LIN {X 0,Y 403.759,Z 485.319,A -85,B 0,C 180,E1 -11073.792,E2 -11073.792} C_VEL
LIN {X 0,Y 400.892,Z 485.679,A -85,B 0,C 180,E1 -11075.141,E2 -11075.141} C_VEL
LIN {X 0,Y 398.47,Z 485.978,A -85,B 0,C 180,E1 -11076.231,E2 -11076.231} C_VEL
LIN {X 0,Y 397.442,Z 486.102,A -85,B 0,C 180,E1 -11077.075,E2 -11077.075} C_VEL
LIN {X 0,Y 397.364,Z 486.11,A -85,B 0,C 180,E1 -11077.36,E2 -11077.36} C_VEL
LIN {X 0,Y 397.201,Z 486.134,A -85,B 0,C 180,E1 -11081.223,E2 -11081.223} C_VEL
LIN {X 0,Y 397.178,Z 486.132,A -85,B 0,C 180,E1 -11084.343,E2 -11084.343} C_VEL
LIN {X 0,Y 397.176,Z 486.138,A -85,B 0,C 180,E1 -11087.507,E2 -11087.507} C_VEL
LIN {X 0,Y 397.11,Z 486.141,A -85,B 0,C 180,E1 -11090.73,E2 -11090.73} C_VEL
LIN {X 0,Y 397.134,Z 486.138,A -85,B 0,C 180,E1 -11094.018,E2 -11094.018} C_VEL
LIN {X 0,Y 397.196,Z 486.137,A -85,B 0,C 180,E1 -11097.39,E2 -11097.39} C_VEL
LIN {X 0,Y 397.08,Z 486.146,A -85,B 0,C 180,E1 -11100.882,E2 -11100.882} C_VEL
LIN {X 0,Y 397.127,Z 486.138,A -85,B 0,C 180,E1 -11104.493,E2 -11104.493} C_VEL
LIN {X 0,Y 397.105,Z 486.141,A -85,B 0,C 180,E1 -11108.275,E2 -11108.275} C_VEL
LIN {X 0,Y 397.092,Z 486.145,A -85,B 0,C 180,E1 -11110.909,E2 -11110.909} C_VEL
LIN {X 0,Y 397.105,Z 486.144,A -85,B 0,C 180,E1 -11113.648,E2 -11113.648} C_VEL
LIN {X 0,Y 397.103,Z 486.141,A -85,B 0,C 180,E1 -11116.521,E2 -11116.521} C_VEL
LIN {X 0,Y 397.115,Z 486.14,A -85,B 0,C 180,E1 -11120.423,E2 -11120.423} C_VEL
LIN {X 0,Y 397.11,Z 486.14,A -85,B 0,C 180,E1 -11124.266,E2 -11124.266} C_VEL
LIN {X 0,Y 397.116,Z 486.141,A -85,B 0,C 180,E1 -11126.727,E2 -11126.727} C_VEL
LIN {X 0,Y 397.188,Z 486.311,A -85,B 0,C 180,E1 -11130.065,E2 -11130.065} C_VEL
LIN {X 0,Y 400.62,Z 501.643,A -85,B 0,C 180,E1 -11132.863,E2 -11132.863} C_VEL
LIN {X 0,Y 401.755,Z 508.389,A -85,B 0,C 180,E1 -11134.066,E2 -11134.066} C_VEL
LIN {X 0,Y 400.796,Z 526.433,A -85,B 0,C 180,E1 -11137.036,E2 -11137.036} C_VEL
LIN {X 0,Y 399.909,Z 544.238,A -85,B 0,C 180,E1 -11139.959,E2 -11139.959} C_VEL
LIN {X 0,Y 399.783,Z 547.353,A -85,B 0,C 180,E1 -11140.471,E2 -11140.471} C_VEL
LIN {X 0,Y 402.807,Z 568.009,A -85,B 0,C 180,E1 -11141.071,E2 -11141.071} C_VEL
LIN {X 0,Y 401.01,Z 658.287,A -85,B 0,C 180,E1 -11143.06,E2 -11143.06} C_VEL
LIN {X 0,Y 400.556,Z 670.536,A -85,B 0,C 180,E1 -11143.5,E2 -11143.5} C_VEL
LIN {X 0,Y 399.98,Z 683.841,A -85,B 0,C 180,E1 -11144.196,E2 -11144.196} C_VEL
LIN {X 0,Y 399.423,Z 695.225,A -85,B 0,C 180,E1 -11144.984,E2 -11144.984} C_VEL
LIN {X 0,Y 398.841,Z 705.755,A -85,B 0,C 180,E1 -11145.901,E2 -11145.901} C_VEL
LIN {X 0,Y 398.184,Z 716.959,A -85,B 0,C 180,E1 -11147.125,E2 -11147.125} C_VEL
LIN {X 0,Y 397.568,Z 725.567,A -85,B 0,C 180,E1 -11148.271,E2 -11148.271} C_VEL
LIN {X 0,Y 397.087,Z 733.527,A -85,B 0,C 180,E1 -11149.548,E2 -11149.548} C_VEL
LIN {X 0,Y 396.575,Z 741.26,A -85,B 0,C 180,E1 -11151.079,E2 -11151.079} C_VEL
LIN {X 0,Y 396.256,Z 746.53,A -85,B 0,C 180,E1 -11152.356,E2 -11152.356} C_VEL
LIN {X 0,Y 396.07,Z 751.606,A -85,B 0,C 180,E1 -11153.888,E2 -11153.888} C_VEL
LIN {X 0,Y 395.925,Z 755.497,A -85,B 0,C 180,E1 -11155.418,E2 -11155.418} C_VEL
LIN {X 0,Y 395.803,Z 758.303,A -85,B 0,C 180,E1 -11156.946,E2 -11156.946} C_VEL
LIN {X 0,Y 395.821,Z 759.622,A -85,B 0,C 180,E1 -11157.965,E2 -11157.965} C_VEL
LIN {X 0,Y 395.796,Z 760.49,A -85,B 0,C 180,E1 -11158.983,E2 -11158.983} C_VEL
LIN {X 0,Y 395.778,Z 760.909,A -85,B 0,C 180,E1 -11160,E2 -11160} C_VEL
LIN {X 0,Y 395.797,Z 760.918,A -85,B 0,C 180,E1 -11161.017,E2 -11161.017} C_VEL
LIN {X 0,Y 395.88,Z 760.496,A -85,B 0,C 180,E1 -11162.035,E2 -11162.035} C_VEL
LIN {X 0,Y 395.894,Z 759.614,A -85,B 0,C 180,E1 -11163.053,E2 -11163.053} C_VEL
LIN {X 0,Y 395.883,Z 758.325,A -85,B 0,C 180,E1 -11164.072,E2 -11164.072} C_VEL
LIN {X 0,Y 396.184,Z 755.531,A -85,B 0,C 180,E1 -11165.599,E2 -11165.599} C_VEL
LIN {X 0,Y 396.413,Z 751.669,A -85,B 0,C 180,E1 -11167.129,E2 -11167.129} C_VEL
LIN {X 0,Y 396.827,Z 745.635,A -85,B 0,C 180,E1 -11168.915,E2 -11168.915} C_VEL
LIN {X 0,Y 397.366,Z 738.969,A -85,B 0,C 180,E1 -11170.445,E2 -11170.445} C_VEL
LIN {X 0,Y 398.091,Z 730.666,A -85,B 0,C 180,E1 -11171.972,E2 -11171.972} C_VEL
LIN {X 0,Y 399.002,Z 720.252,A -85,B 0,C 180,E1 -11173.496,E2 -11173.496} C_VEL
LIN {X 0,Y 399.826,Z 710.965,A -85,B 0,C 180,E1 -11174.595,E2 -11174.595} C_VEL
LIN {X 0,Y 400.649,Z 700,A -85,B 0,C 180,E1 -11175.647,E2 -11175.647} C_VEL
LIN {X 0,Y 401.33,Z 688.464,A -85,B 0,C 180,E1 -11176.533,E2 -11176.533} C_VEL
LIN {X 0,Y 402.167,Z 675.458,A -85,B 0,C 180,E1 -11177.282,E2 -11177.282} C_VEL
LIN {X 0,Y 402.796,Z 661.803,A -85,B 0,C 180,E1 -11177.844,E2 -11177.844} C_VEL
LIN {X 0,Y 403.528,Z 637.136,A -85,B 0,C 180,E1 -11178.467,E2 -11178.467} C_VEL
LIN {X 0,Y 405.694,Z 568.492,A -85,B 0,C 180,E1 -11180.17,E2 -11180.17} C_VEL
LIN {X 0,Y 403.291,Z 554.459,A -85,B 0,C 180,E1 -11180.763,E2 -11180.763} C_VEL
LIN {X 0,Y 402.088,Z 549.119,A -85,B 0,C 180,E1 -11181.03,E2 -11181.03} C_VEL
LIN {X 0,Y 403.433,Z 528.468,A -85,B 0,C 180,E1 -11184.44,E2 -11184.44} C_VEL
LIN {X 0,Y 404.51,Z 513.97,A -85,B 0,C 180,E1 -11186.855,E2 -11186.855} C_VEL
LIN {X 0,Y 403.351,Z 506.568,A -85,B 0,C 180,E1 -11188.256,E2 -11188.256} C_VEL
LIN {X 0,Y 400.855,Z 497.27,A -85,B 0,C 180,E1 -11190.194,E2 -11190.194} C_VEL
LIN {X 0,Y 398.092,Z 489.021,A -85,B 0,C 180,E1 -11192.069,E2 -11192.069} C_VEL
LIN {X 0,Y 397.109,Z 486.15,A -85,B 0,C 180,E1 -11192.782,E2 -11192.782} C_VEL
LIN {X 0,Y 397.11,Z 486.145,A -85,B 0,C 180,E1 -11195.735,E2 -11195.735} C_VEL
LIN {X 0,Y 397.116,Z 486.144,A -85,B 0,C 180,E1 -11199.577,E2 -11199.577} C_VEL
LIN {X 0,Y 397.104,Z 486.142,A -85,B 0,C 180,E1 -11203.479,E2 -11203.479} C_VEL
LIN {X 0,Y 397.108,Z 486.146,A -85,B 0,C 180,E1 -11206.52,E2 -11206.52} C_VEL
LIN {X 0,Y 397.117,Z 486.142,A -85,B 0,C 180,E1 -11209.552,E2 -11209.552} C_VEL
LIN {X 0,Y 397.099,Z 486.144,A -85,B 0,C 180,E1 -11212.79,E2 -11212.79} C_VEL
LIN {X 0,Y 397.12,Z 486.142,A -85,B 0,C 180,E1 -11216.282,E2 -11216.282} C_VEL
LIN {X 0,Y 397.156,Z 486.306,A -85,B 0,C 180,E1 -11219.271,E2 -11219.271} C_VEL
LIN {X 0,Y 401.317,Z 503.352,A -85,B 0,C 180,E1 -11222.632,E2 -11222.632} C_VEL
LIN {X 0,Y 403.042,Z 511.399,A -85,B 0,C 180,E1 -11224.155,E2 -11224.155} C_VEL
LIN {X 0,Y 401.75,Z 526.092,A -85,B 0,C 180,E1 -11226.621,E2 -11226.621} C_VEL
LIN {X 0,Y 405.305,Z 550.044,A -85,B 0,C 180,E1 -11227.331,E2 -11227.331} C_VEL
LIN {X 0,Y 402.877,Z 662.659,A -85,B 0,C 180,E1 -11229.714,E2 -11229.714} C_VEL
LIN {X 0,Y 402.185,Z 677.653,A -85,B 0,C 180,E1 -11230.243,E2 -11230.243} C_VEL
LIN {X 0,Y 401.574,Z 691,A -85,B 0,C 180,E1 -11230.92,E2 -11230.92} C_VEL
LIN {X 0,Y 400.808,Z 703.38,A -85,B 0,C 180,E1 -11231.734,E2 -11231.734} C_VEL
LIN {X 0,Y 399.927,Z 715.719,A -85,B 0,C 180,E1 -11232.75,E2 -11232.75} C_VEL
LIN {X 0,Y 399.03,Z 727.035,A -85,B 0,C 180,E1 -11233.895,E2 -11233.895} C_VEL
LIN {X 0,Y 398.233,Z 737.447,A -85,B 0,C 180,E1 -11235.173,E2 -11235.173} C_VEL
LIN {X 0,Y 397.446,Z 747.737,A -85,B 0,C 180,E1 -11236.71,E2 -11236.71} C_VEL
LIN {X 0,Y 396.938,Z 756.248,A -85,B 0,C 180,E1 -11238.252,E2 -11238.252} C_VEL
LIN {X 0,Y 396.373,Z 764.324,A -85,B 0,C 180,E1 -11240.045,E2 -11240.045} C_VEL
LIN {X 0,Y 396.054,Z 770.763,A -85,B 0,C 180,E1 -11241.839,E2 -11241.839} C_VEL
LIN {X 0,Y 395.859,Z 776.269,A -85,B 0,C 180,E1 -11243.833,E2 -11243.833} C_VEL
LIN {X 0,Y 395.825,Z 778.539,A -85,B 0,C 180,E1 -11244.907,E2 -11244.907} C_VEL
LIN {X 0,Y 395.73,Z 781.666,A -85,B 0,C 180,E1 -11246.946,E2 -11246.946} C_VEL
LIN {X 0,Y 395.817,Z 782.675,A -85,B 0,C 180,E1 -11247.965,E2 -11247.965} C_VEL
LIN {X 0,Y 395.777,Z 783.588,A -85,B 0,C 180,E1 -11250,E2 -11250} C_VEL
LIN {X 0,Y 395.785,Z 783.048,A -85,B 0,C 180,E1 -11252.035,E2 -11252.035} C_VEL
LIN {X 0,Y 395.764,Z 781.056,A -85,B 0,C 180,E1 -11254.073,E2 -11254.073} C_VEL
LIN {X 0,Y 395.861,Z 777.535,A -85,B 0,C 180,E1 -11256.115,E2 -11256.115} C_VEL
LIN {X 0,Y 396.01,Z 773.868,A -85,B 0,C 180,E1 -11257.649,E2 -11257.649} C_VEL
LIN {X 0,Y 396.267,Z 769.217,A -85,B 0,C 180,E1 -11259.185,E2 -11259.185} C_VEL
LIN {X 0,Y 396.729,Z 762.473,A -85,B 0,C 180,E1 -11260.978,E2 -11260.978} C_VEL
LIN {X 0,Y 397.438,Z 754.082,A -85,B 0,C 180,E1 -11262.77,E2 -11262.77} C_VEL
LIN {X 0,Y 398.202,Z 745.265,A -85,B 0,C 180,E1 -11264.306,E2 -11264.306} C_VEL
LIN {X 0,Y 399.099,Z 734.56,A -85,B 0,C 180,E1 -11265.84,E2 -11265.84} C_VEL
LIN {X 0,Y 400.301,Z 722.607,A -85,B 0,C 180,E1 -11267.234,E2 -11267.234} C_VEL
LIN {X 0,Y 401.354,Z 710.635,A -85,B 0,C 180,E1 -11268.373,E2 -11268.373} C_VEL
LIN {X 0,Y 402.487,Z 697.45,A -85,B 0,C 180,E1 -11269.376,E2 -11269.376} C_VEL
LIN {X 0,Y 403.457,Z 683.624,A -85,B 0,C 180,E1 -11270.189,E2 -11270.189} C_VEL
LIN {X 0,Y 404.256,Z 670.939,A -85,B 0,C 180,E1 -11270.746,E2 -11270.746} C_VEL
LIN {X 0,Y 404.865,Z 655.605,A -85,B 0,C 180,E1 -11271.212,E2 -11271.212} C_VEL
LIN {X 0,Y 407.382,Z 577.138,A -85,B 0,C 180,E1 -11273.008,E2 -11273.008} C_VEL
LIN {X 0,Y 408.254,Z 550.433,A -85,B 0,C 180,E1 -11273.667,E2 -11273.667} C_VEL
LIN {X 0,Y 406.388,Z 537.955,A -85,B 0,C 180,E1 -11274.177,E2 -11274.177} C_VEL
LIN {X 0,Y 404.344,Z 528.079,A -85,B 0,C 180,E1 -11274.655,E2 -11274.655} C_VEL
LIN {X 0,Y 405.873,Z 518.481,A -85,B 0,C 180,E1 -11276.48,E2 -11276.48} C_VEL
LIN {X 0,Y 404.372,Z 509.978,A -85,B 0,C 180,E1 -11278.552,E2 -11278.552} C_VEL
LIN {X 0,Y 402.351,Z 502.415,A -85,B 0,C 180,E1 -11280.688,E2 -11280.688} C_VEL
LIN {X 0,Y 400.233,Z 495.392,A -85,B 0,C 180,E1 -11282.981,E2 -11282.981} C_VEL
LIN {X 0,Y 398.482,Z 490.292,A -85,B 0,C 180,E1 -11284.974,E2 -11284.974} C_VEL
LIN {X 0,Y 397.118,Z 486.145,A -85,B 0,C 180,E1 -11286.914,E2 -11286.914} C_VEL
LIN {X 0,Y 397.116,Z 486.145,A -85,B 0,C 180,E1 -11289.577,E2 -11289.577} C_VEL
LIN {X 0,Y 397.107,Z 486.145,A -85,B 0,C 180,E1 -11293.48,E2 -11293.48} C_VEL
LIN {X 0,Y 397.105,Z 486.146,A -85,B 0,C 180,E1 -11296.521,E2 -11296.521} C_VEL
LIN {X 0,Y 397.116,Z 486.145,A -85,B 0,C 180,E1 -11300.423,E2 -11300.423} C_VEL
LIN {X 0,Y 397.133,Z 486.272,A -85,B 0,C 180,E1 -11304.033,E2 -11304.033} C_VEL
LIN {X 0,Y 399.278,Z 492.635,A -85,B 0,C 180,E1 -11306.931,E2 -11306.931} C_VEL
LIN {X 0,Y 401.371,Z 499.612,A -85,B 0,C 180,E1 -11309.483,E2 -11309.483} C_VEL
LIN {X 0,Y 403.453,Z 507.524,A -85,B 0,C 180,E1 -11311.944,E2 -11311.944} C_VEL
LIN {X 0,Y 404.967,Z 516.192,A -85,B 0,C 180,E1 -11314.287,E2 -11314.287} C_VEL
LIN {X 0,Y 402.804,Z 531.826,A -85,B 0,C 180,E1 -11317.628,E2 -11317.628} C_VEL
LIN {X 0,Y 402.05,Z 539.246,A -85,B 0,C 180,E1 -11319.116,E2 -11319.116} C_VEL
LIN {X 0,Y 405.319,Z 554.337,A -85,B 0,C 180,E1 -11319.895,E2 -11319.895} C_VEL
LIN {X 0,Y 407.27,Z 567.227,A -85,B 0,C 180,E1 -11320.467,E2 -11320.467} C_VEL
LIN {X 0,Y 404.15,Z 643.587,A -85,B 0,C 180,E1 -11322.479,E2 -11322.479} C_VEL
LIN {X 0,Y 403.473,Z 659.097,A -85,B 0,C 180,E1 -11322.939,E2 -11322.939} C_VEL
LIN {X 0,Y 402.655,Z 673.328,A -85,B 0,C 180,E1 -11323.588,E2 -11323.588} C_VEL
LIN {X 0,Y 401.957,Z 685.093,A -85,B 0,C 180,E1 -11324.31,E2 -11324.31} C_VEL
LIN {X 0,Y 400.993,Z 697.434,A -85,B 0,C 180,E1 -11325.278,E2 -11325.278} C_VEL
LIN {X 0,Y 399.992,Z 708.895,A -85,B 0,C 180,E1 -11326.408,E2 -11326.408} C_VEL
LIN {X 0,Y 399.132,Z 718.272,A -85,B 0,C 180,E1 -11327.543,E2 -11327.543} C_VEL
LIN {X 0,Y 398.416,Z 726.885,A -85,B 0,C 180,E1 -11328.811,E2 -11328.811} C_VEL
LIN {X 0,Y 397.585,Z 735.348,A -85,B 0,C 180,E1 -11330.333,E2 -11330.333} C_VEL
LIN {X 0,Y 396.962,Z 742.204,A -85,B 0,C 180,E1 -11331.857,E2 -11331.857} C_VEL
LIN {X 0,Y 396.653,Z 747.66,A -85,B 0,C 180,E1 -11333.387,E2 -11333.387} C_VEL
LIN {X 0,Y 396.145,Z 751.925,A -85,B 0,C 180,E1 -11334.911,E2 -11334.911} C_VEL
LIN {X 0,Y 396.195,Z 754.147,A -85,B 0,C 180,E1 -11335.931,E2 -11335.931} C_VEL
LIN {X 0,Y 396.076,Z 755.88,A -85,B 0,C 180,E1 -11336.949,E2 -11336.949} C_VEL
LIN {X 0,Y 395.911,Z 757.195,A -85,B 0,C 180,E1 -11337.965,E2 -11337.965} C_VEL
LIN {X 0,Y 395.817,Z 758.093,A -85,B 0,C 180,E1 -11338.983,E2 -11338.983} C_VEL
LIN {X 0,Y 395.779,Z 758.541,A -85,B 0,C 180,E1 -11340,E2 -11340} C_VEL
LIN {X 0,Y 395.796,Z 758.548,A -85,B 0,C 180,E1 -11341.017,E2 -11341.017} C_VEL
LIN {X 0,Y 395.835,Z 758.142,A -85,B 0,C 180,E1 -11342.035,E2 -11342.035} C_VEL
LIN {X 0,Y 395.803,Z 757.324,A -85,B 0,C 180,E1 -11343.054,E2 -11343.054} C_VEL
LIN {X 0,Y 395.823,Z 756.036,A -85,B 0,C 180,E1 -11344.073,E2 -11344.073} C_VEL
LIN {X 0,Y 395.945,Z 753.287,A -85,B 0,C 180,E1 -11345.602,E2 -11345.602} C_VEL
LIN {X 0,Y 396.06,Z 749.463,A -85,B 0,C 180,E1 -11347.135,E2 -11347.135} C_VEL
LIN {X 0,Y 396.329,Z 744.458,A -85,B 0,C 180,E1 -11348.669,E2 -11348.669} C_VEL
LIN {X 0,Y 396.697,Z 738.131,A -85,B 0,C 180,E1 -11350.205,E2 -11350.205} C_VEL
LIN {X 0,Y 397.221,Z 730.26,A -85,B 0,C 180,E1 -11351.74,E2 -11351.74} C_VEL
LIN {X 0,Y 397.719,Z 722.24,A -85,B 0,C 180,E1 -11353.021,E2 -11353.021} C_VEL
LIN {X 0,Y 398.35,Z 712.484,A -85,B 0,C 180,E1 -11354.3,E2 -11354.3} C_VEL
LIN {X 0,Y 399.064,Z 701.717,A -85,B 0,C 180,E1 -11355.448,E2 -11355.448} C_VEL
LIN {X 0,Y 399.854,Z 689.869,A -85,B 0,C 180,E1 -11356.464,E2 -11356.464} C_VEL
LIN {X 0,Y 400.489,Z 677.457,A -85,B 0,C 180,E1 -11357.291,E2 -11357.291} C_VEL
LIN {X 0,Y 401.065,Z 663.404,A -85,B 0,C 180,E1 -11357.99,E2 -11357.99} C_VEL
LIN {X 0,Y 401.569,Z 650.05,A -85,B 0,C 180,E1 -11358.428,E2 -11358.428} C_VEL
LIN {X 0,Y 403.507,Z 565.666,A -85,B 0,C 180,E1 -11360.332,E2 -11360.332} C_VEL
LIN {X 0,Y 399.716,Z 540.055,A -85,B 0,C 180,E1 -11361.132,E2 -11361.132} C_VEL
LIN {X 0,Y 401.088,Z 521.32,A -85,B 0,C 180,E1 -11364.666,E2 -11364.666} C_VEL
LIN {X 0,Y 402.077,Z 508.941,A -85,B 0,C 180,E1 -11367.03,E2 -11367.03} C_VEL
LIN {X 0,Y 399.623,Z 497.259,A -85,B 0,C 180,E1 -11369.5,E2 -11369.5} C_VEL
LIN {X 0,Y 397.092,Z 486.149,A -85,B 0,C 180,E1 -11371.947,E2 -11371.947} C_VEL
LIN {X 0,Y 397.128,Z 486.142,A -85,B 0,C 180,E1 -11374.493,E2 -11374.493} C_VEL
LIN {X 0,Y 397.109,Z 486.141,A -85,B 0,C 180,E1 -11378.274,E2 -11378.274} C_VEL
LIN {X 0,Y 397.092,Z 486.143,A -85,B 0,C 180,E1 -11380.908,E2 -11380.908} C_VEL
LIN {X 0,Y 397.103,Z 486.148,A -85,B 0,C 180,E1 -11383.648,E2 -11383.648} C_VEL
LIN {X 0,Y 397.104,Z 486.141,A -85,B 0,C 180,E1 -11386.521,E2 -11386.521} C_VEL
LIN {X 0,Y 397.114,Z 486.14,A -85,B 0,C 180,E1 -11390.423,E2 -11390.423} C_VEL
LIN {X 0,Y 397.11,Z 486.141,A -85,B 0,C 180,E1 -11394.265,E2 -11394.265} C_VEL
LIN {X 0,Y 397.116,Z 486.14,A -85,B 0,C 180,E1 -11396.727,E2 -11396.727} C_VEL
LIN {X 0,Y 397.126,Z 486.139,A -85,B 0,C 180,E1 -11400.296,E2 -11400.296} C_VEL
LIN {X 0,Y 397.196,Z 486.129,A -85,B 0,C 180,E1 -11402.61,E2 -11402.61} C_VEL
LIN {X 0,Y 397.135,Z 486.139,A -85,B 0,C 180,E1 -11405.982,E2 -11405.982} C_VEL
LIN {X 0,Y 397.146,Z 486.141,A -85,B 0,C 180,E1 -11409.702,E2 -11409.702} C_VEL
LIN {X 0,Y 397.183,Z 486.132,A -85,B 0,C 180,E1 -11412.845,E2 -11412.845} C_VEL
LIN {X 0,Y 397.228,Z 486.126,A -85,B 0,C 180,E1 -11416.679,E2 -11416.679} C_VEL
LIN {X 0,Y 397.22,Z 486.13,A -85,B 0,C 180,E1 -11419.809,E2 -11419.809} C_VEL
LIN {X 0,Y 397.366,Z 486.11,A -85,B 0,C 180,E1 -11422.888,E2 -11422.888} C_VEL
LIN {X 0,Y 397.257,Z 486.123,A -85,B 0,C 180,E1 -11424.925,E2 -11424.925} C_VEL
LIN {X 0,Y 397.453,Z 486.099,A -85,B 0,C 180,E1 -11427.973,E2 -11427.973} C_VEL
LIN {X 0,Y 397.583,Z 486.083,A -85,B 0,C 180,E1 -11430,E2 -11430} C_VEL
LIN {X 0,Y 397.384,Z 486.109,A -85,B 0,C 180,E1 -11433.041,E2 -11433.041} C_VEL
LIN {X 0,Y 397.364,Z 486.112,A -85,B 0,C 180,E1 -11437.112,E2 -11437.112} C_VEL
LIN {X 0,Y 397.364,Z 486.11,A -85,B 0,C 180,E1 -11437.36,E2 -11437.36} C_VEL
LIN {X 0,Y 396.694,Z 486.193,A -85,B 0,C 180,E1 -11438.206,E2 -11438.206} C_VEL
LIN {X 0,Y 393.768,Z 486.562,A -85,B 0,C 180,E1 -11439.578,E2 -11439.578} C_VEL
LIN {X 0,Y 391.285,Z 486.873,A -85,B 0,C 180,E1 -11440.686,E2 -11440.686} C_VEL
LIN {X 0,Y 390.226,Z 487.003,A -85,B 0,C 180,E1 -11441.545,E2 -11441.545} C_VEL
LIN {X 0,Y 390.143,Z 487.01,A -85,B 0,C 180,E1 -11441.836,E2 -11441.836} C_VEL
LIN {X 0,Y 390.146,Z 487.008,A -85,B 0,C 180,E1 -11444.607,E2 -11444.607} C_VEL
LIN {X 0,Y 390.129,Z 487.012,A -85,B 0,C 180,E1 -11447.833,E2 -11447.833} C_VEL
LIN {X 0,Y 390.064,Z 487.022,A -85,B 0,C 180,E1 -11451.122,E2 -11451.122} C_VEL
LIN {X 0,Y 390.081,Z 487.016,A -85,B 0,C 180,E1 -11454.481,E2 -11454.481} C_VEL
LIN {X 0,Y 390.118,Z 487.012,A -85,B 0,C 180,E1 -11457.93,E2 -11457.93} C_VEL
LIN {X 0,Y 390.025,Z 487.028,A -85,B 0,C 180,E1 -11461.504,E2 -11461.504} C_VEL
LIN {X 0,Y 390.086,Z 487.021,A -85,B 0,C 180,E1 -11465.207,E2 -11465.207} C_VEL
LIN {X 0,Y 390.072,Z 487.023,A -85,B 0,C 180,E1 -11469.219,E2 -11469.219} C_VEL
LIN {X 0,Y 390.046,Z 487.02,A -85,B 0,C 180,E1 -11472.375,E2 -11472.375} C_VEL
LIN {X 0,Y 390.047,Z 487.027,A -85,B 0,C 180,E1 -11475.355,E2 -11475.355} C_VEL
LIN {X 0,Y 390.032,Z 487.022,A -85,B 0,C 180,E1 -11478.187,E2 -11478.187} C_VEL
LIN {X 0,Y 390.091,Z 487.017,A -85,B 0,C 180,E1 -11480.908,E2 -11480.908} C_VEL
LIN {X 0,Y 390.087,Z 487.017,A -85,B 0,C 180,E1 -11484.793,E2 -11484.793} C_VEL
LIN {X 0,Y 390.029,Z 487.025,A -85,B 0,C 180,E1 -11488.496,E2 -11488.496} C_VEL
LIN {X 0,Y 390.096,Z 487.037,A -85,B 0,C 180,E1 -11489.768,E2 -11489.768} C_VEL
LIN {X 0,Y 393.774,Z 503.467,A -85,B 0,C 180,E1 -11492.797,E2 -11492.797} C_VEL
LIN {X 0,Y 394.854,Z 509.388,A -85,B 0,C 180,E1 -11493.863,E2 -11493.863} C_VEL
LIN {X 0,Y 393.877,Z 527.561,A -85,B 0,C 180,E1 -11496.887,E2 -11496.887} C_VEL
LIN {X 0,Y 392.947,Z 545.481,A -85,B 0,C 180,E1 -11499.861,E2 -11499.861} C_VEL
LIN {X 0,Y 392.838,Z 547.511,A -85,B 0,C 180,E1 -11500.195,E2 -11500.195} C_VEL
LIN {X 0,Y 395.918,Z 569.818,A -85,B 0,C 180,E1 -11500.852,E2 -11500.852} C_VEL
LIN {X 0,Y 394.066,Z 658.396,A -85,B 0,C 180,E1 -11502.853,E2 -11502.853} C_VEL
LIN {X 0,Y 393.575,Z 671.35,A -85,B 0,C 180,E1 -11503.332,E2 -11503.332} C_VEL
LIN {X 0,Y 392.986,Z 684.47,A -85,B 0,C 180,E1 -11504.04,E2 -11504.04} C_VEL
LIN {X 0,Y 392.323,Z 697.027,A -85,B 0,C 180,E1 -11504.945,E2 -11504.945} C_VEL
LIN {X 0,Y 391.769,Z 707.595,A -85,B 0,C 180,E1 -11505.919,E2 -11505.919} C_VEL
LIN {X 0,Y 391.096,Z 718.444,A -85,B 0,C 180,E1 -11507.151,E2 -11507.151} C_VEL
LIN {X 0,Y 390.341,Z 728.482,A -85,B 0,C 180,E1 -11508.577,E2 -11508.577} C_VEL
LIN {X 0,Y 389.773,Z 737.331,A -85,B 0,C 180,E1 -11510.137,E2 -11510.137} C_VEL
LIN {X 0,Y 389.313,Z 744.357,A -85,B 0,C 180,E1 -11511.696,E2 -11511.696} C_VEL
LIN {X 0,Y 389.05,Z 750.711,A -85,B 0,C 180,E1 -11513.49,E2 -11513.49} C_VEL
LIN {X 0,Y 388.906,Z 754.32,A -85,B 0,C 180,E1 -11514.816,E2 -11514.816} C_VEL
LIN {X 0,Y 388.784,Z 756.607,A -85,B 0,C 180,E1 -11515.853,E2 -11515.853} C_VEL
LIN {X 0,Y 388.708,Z 758.378,A -85,B 0,C 180,E1 -11516.891,E2 -11516.891} C_VEL
LIN {X 0,Y 388.72,Z 759.725,A -85,B 0,C 180,E1 -11517.928,E2 -11517.928} C_VEL
LIN {X 0,Y 388.709,Z 760.648,A -85,B 0,C 180,E1 -11518.964,E2 -11518.964} C_VEL
LIN {X 0,Y 388.708,Z 761.098,A -85,B 0,C 180,E1 -11520,E2 -11520} C_VEL
LIN {X 0,Y 388.729,Z 761.137,A -85,B 0,C 180,E1 -11521.036,E2 -11521.036} C_VEL
LIN {X 0,Y 388.797,Z 760.762,A -85,B 0,C 180,E1 -11522.072,E2 -11522.072} C_VEL
LIN {X 0,Y 388.801,Z 759.919,A -85,B 0,C 180,E1 -11523.109,E2 -11523.109} C_VEL
LIN {X 0,Y 388.809,Z 758.653,A -85,B 0,C 180,E1 -11524.146,E2 -11524.146} C_VEL
LIN {X 0,Y 389.143,Z 755.903,A -85,B 0,C 180,E1 -11525.701,E2 -11525.701} C_VEL
LIN {X 0,Y 389.381,Z 752.083,A -85,B 0,C 180,E1 -11527.258,E2 -11527.258} C_VEL
LIN {X 0,Y 389.753,Z 747.077,A -85,B 0,C 180,E1 -11528.817,E2 -11528.817} C_VEL
LIN {X 0,Y 390.332,Z 740.755,A -85,B 0,C 180,E1 -11530.373,E2 -11530.373} C_VEL
LIN {X 0,Y 391.05,Z 732.834,A -85,B 0,C 180,E1 -11531.928,E2 -11531.928} C_VEL
LIN {X 0,Y 391.817,Z 724.751,A -85,B 0,C 180,E1 -11533.22,E2 -11533.22} C_VEL
LIN {X 0,Y 392.717,Z 714.89,A -85,B 0,C 180,E1 -11534.51,E2 -11534.51} C_VEL
LIN {X 0,Y 393.659,Z 703.857,A -85,B 0,C 180,E1 -11535.666,E2 -11535.666} C_VEL
LIN {X 0,Y 394.478,Z 691.597,A -85,B 0,C 180,E1 -11536.695,E2 -11536.695} C_VEL
LIN {X 0,Y 395.453,Z 678.541,A -85,B 0,C 180,E1 -11537.519,E2 -11537.519} C_VEL
LIN {X 0,Y 396.137,Z 665.425,A -85,B 0,C 180,E1 -11538.121,E2 -11538.121} C_VEL
LIN {X 0,Y 396.621,Z 651.921,A -85,B 0,C 180,E1 -11538.533,E2 -11538.533} C_VEL
LIN {X 0,Y 399.163,Z 580.325,A -85,B 0,C 180,E1 -11540.334,E2 -11540.334} C_VEL
LIN {X 0,Y 399.413,Z 569.52,A -85,B 0,C 180,E1 -11540.631,E2 -11540.631} C_VEL
LIN {X 0,Y 397.174,Z 556.201,A -85,B 0,C 180,E1 -11541.217,E2 -11541.217} C_VEL
LIN {X 0,Y 395.628,Z 549.275,A -85,B 0,C 180,E1 -11541.595,E2 -11541.595} C_VEL
LIN {X 0,Y 397.044,Z 529.798,A -85,B 0,C 180,E1 -11544.86,E2 -11544.86} C_VEL
LIN {X 0,Y 398.07,Z 516.818,A -85,B 0,C 180,E1 -11547.041,E2 -11547.041} C_VEL
LIN {X 0,Y 397.353,Z 510.777,A -85,B 0,C 180,E1 -11548.225,E2 -11548.225} C_VEL
LIN {X 0,Y 395.155,Z 502.052,A -85,B 0,C 180,E1 -11550.069,E2 -11550.069} C_VEL
LIN {X 0,Y 392.283,Z 493.041,A -85,B 0,C 180,E1 -11552.165,E2 -11552.165} C_VEL
LIN {X 0,Y 390.076,Z 487.024,A -85,B 0,C 180,E1 -11553.721,E2 -11553.721} C_VEL
LIN {X 0,Y 390.059,Z 487.025,A -85,B 0,C 180,E1 -11556.483,E2 -11556.483} C_VEL
LIN {X 0,Y 390.072,Z 487.022,A -85,B 0,C 180,E1 -11559.218,E2 -11559.218} C_VEL
LIN {X 0,Y 390.044,Z 487.023,A -85,B 0,C 180,E1 -11562.374,E2 -11562.374} C_VEL
LIN {X 0,Y 390.048,Z 487.021,A -85,B 0,C 180,E1 -11565.355,E2 -11565.355} C_VEL
LIN {X 0,Y 390.069,Z 487.023,A -85,B 0,C 180,E1 -11568.192,E2 -11568.192} C_VEL
LIN {X 0,Y 390.094,Z 487.016,A -85,B 0,C 180,E1 -11570.908,E2 -11570.908} C_VEL
LIN {X 0,Y 390.087,Z 487.018,A -85,B 0,C 180,E1 -11574.793,E2 -11574.793} C_VEL
LIN {X 0,Y 390.066,Z 487.025,A -85,B 0,C 180,E1 -11578.499,E2 -11578.499} C_VEL
LIN {X 0,Y 390.092,Z 487.14,A -85,B 0,C 180,E1 -11578.917,E2 -11578.917} C_VEL
LIN {X 0,Y 394.295,Z 504.428,A -85,B 0,C 180,E1 -11582.391,E2 -11582.391} C_VEL
LIN {X 0,Y 396.091,Z 512.51,A -85,B 0,C 180,E1 -11583.95,E2 -11583.95} C_VEL
LIN {X 0,Y 395.629,Z 519.104,A -85,B 0,C 180,E1 -11585.086,E2 -11585.086} C_VEL
LIN {X 0,Y 394.918,Z 526.239,A -85,B 0,C 180,E1 -11586.299,E2 -11586.299} C_VEL
LIN {X 0,Y 398.564,Z 551.351,A -85,B 0,C 180,E1 -11587.054,E2 -11587.054} C_VEL
LIN {X 0,Y 396.021,Z 661.858,A -85,B 0,C 180,E1 -11589.449,E2 -11589.449} C_VEL
LIN {X 0,Y 395.353,Z 676.281,A -85,B 0,C 180,E1 -11589.955,E2 -11589.955} C_VEL
LIN {X 0,Y 394.668,Z 690.559,A -85,B 0,C 180,E1 -11590.68,E2 -11590.68} C_VEL
LIN {X 0,Y 393.853,Z 703.362,A -85,B 0,C 180,E1 -11591.534,E2 -11591.534} C_VEL
LIN {X 0,Y 392.944,Z 715.676,A -85,B 0,C 180,E1 -11592.567,E2 -11592.567} C_VEL
LIN {X 0,Y 391.94,Z 728.078,A -85,B 0,C 180,E1 -11593.863,E2 -11593.863} C_VEL
LIN {X 0,Y 391.131,Z 738.288,A -85,B 0,C 180,E1 -11595.164,E2 -11595.164} C_VEL
LIN {X 0,Y 390.367,Z 748.424,A -85,B 0,C 180,E1 -11596.73,E2 -11596.73} C_VEL
LIN {X 0,Y 389.822,Z 756.793,A -85,B 0,C 180,E1 -11598.298,E2 -11598.298} C_VEL
LIN {X 0,Y 389.281,Z 764.746,A -85,B 0,C 180,E1 -11600.124,E2 -11600.124} C_VEL
LIN {X 0,Y 388.978,Z 770.231,A -85,B 0,C 180,E1 -11601.689,E2 -11601.689} C_VEL
LIN {X 0,Y 388.818,Z 774.667,A -85,B 0,C 180,E1 -11603.253,E2 -11603.253} C_VEL
LIN {X 0,Y 388.724,Z 778.151,A -85,B 0,C 180,E1 -11604.814,E2 -11604.814} C_VEL
LIN {X 0,Y 388.637,Z 781.339,A -85,B 0,C 180,E1 -11606.89,E2 -11606.89} C_VEL
LIN {X 0,Y 388.715,Z 782.375,A -85,B 0,C 180,E1 -11607.928,E2 -11607.928} C_VEL
LIN {X 0,Y 388.706,Z 783.339,A -85,B 0,C 180,E1 -11610,E2 -11610} C_VEL
LIN {X 0,Y 388.723,Z 783.273,A -85,B 0,C 180,E1 -11611.036,E2 -11611.036} C_VEL
LIN {X 0,Y 388.63,Z 782.047,A -85,B 0,C 180,E1 -11613.11,E2 -11613.11} C_VEL
LIN {X 0,Y 388.687,Z 780.891,A -85,B 0,C 180,E1 -11614.148,E2 -11614.148} C_VEL
LIN {X 0,Y 388.797,Z 777.427,A -85,B 0,C 180,E1 -11616.227,E2 -11616.227} C_VEL
LIN {X 0,Y 388.943,Z 773.775,A -85,B 0,C 180,E1 -11617.789,E2 -11617.789} C_VEL
LIN {X 0,Y 389.237,Z 769.163,A -85,B 0,C 180,E1 -11619.352,E2 -11619.352} C_VEL
LIN {X 0,Y 389.709,Z 762.466,A -85,B 0,C 180,E1 -11621.179,E2 -11621.179} C_VEL
LIN {X 0,Y 390.463,Z 754.128,A -85,B 0,C 180,E1 -11623.002,E2 -11623.002} C_VEL
LIN {X 0,Y 391.287,Z 745.389,A -85,B 0,C 180,E1 -11624.564,E2 -11624.564} C_VEL
LIN {X 0,Y 392.27,Z 734.765,A -85,B 0,C 180,E1 -11626.123,E2 -11626.123} C_VEL
LIN {X 0,Y 393.527,Z 722.921,A -85,B 0,C 180,E1 -11627.54,E2 -11627.54} C_VEL
LIN {X 0,Y 394.635,Z 711.088,A -85,B 0,C 180,E1 -11628.697,E2 -11628.697} C_VEL
LIN {X 0,Y 395.845,Z 698.143,A -85,B 0,C 180,E1 -11629.715,E2 -11629.715} C_VEL
LIN {X 0,Y 396.861,Z 684.686,A -85,B 0,C 180,E1 -11630.54,E2 -11630.54} C_VEL
LIN {X 0,Y 397.745,Z 671.699,A -85,B 0,C 180,E1 -11631.135,E2 -11631.135} C_VEL
LIN {X 0,Y 398.428,Z 657.03,A -85,B 0,C 180,E1 -11631.606,E2 -11631.606} C_VEL
LIN {X 0,Y 401.187,Z 577.467,A -85,B 0,C 180,E1 -11633.496,E2 -11633.496} C_VEL
LIN {X 0,Y 402.127,Z 551.327,A -85,B 0,C 180,E1 -11634.164,E2 -11634.164} C_VEL
LIN {X 0,Y 400.294,Z 538.911,A -85,B 0,C 180,E1 -11634.699,E2 -11634.699} C_VEL
LIN {X 0,Y 398.049,Z 528.374,A -85,B 0,C 180,E1 -11635.242,E2 -11635.242} C_VEL
LIN {X 0,Y 399.321,Z 521.087,A -85,B 0,C 180,E1 -11636.667,E2 -11636.667} C_VEL
LIN {X 0,Y 398.44,Z 515.124,A -85,B 0,C 180,E1 -11638.123,E2 -11638.123} C_VEL
LIN {X 0,Y 396.537,Z 507.219,A -85,B 0,C 180,E1 -11640.339,E2 -11640.339} C_VEL
LIN {X 0,Y 394.159,Z 498.992,A -85,B 0,C 180,E1 -11643.067,E2 -11643.067} C_VEL
LIN {X 0,Y 392.061,Z 492.585,A -85,B 0,C 180,E1 -11645.708,E2 -11645.708} C_VEL
LIN {X 0,Y 390.565,Z 488.947,A -85,B 0,C 180,E1 -11647.65,E2 -11647.65} C_VEL
LIN {X 0,Y 390.086,Z 487.02,A -85,B 0,C 180,E1 -11648.844,E2 -11648.844} C_VEL
LIN {X 0,Y 390.047,Z 487.024,A -85,B 0,C 180,E1 -11652.375,E2 -11652.375} C_VEL
LIN {X 0,Y 390.048,Z 487.024,A -85,B 0,C 180,E1 -11655.355,E2 -11655.355} C_VEL
LIN {X 0,Y 390.033,Z 487.026,A -85,B 0,C 180,E1 -11658.187,E2 -11658.187} C_VEL
LIN {X 0,Y 390.071,Z 487.023,A -85,B 0,C 180,E1 -11661.567,E2 -11661.567} C_VEL
LIN {X 0,Y 390.104,Z 487.29,A -85,B 0,C 180,E1 -11662.227,E2 -11662.227} C_VEL
LIN {X 0,Y 391.326,Z 490.926,A -85,B 0,C 180,E1 -11664.371,E2 -11664.371} C_VEL
LIN {X 0,Y 392.78,Z 494.961,A -85,B 0,C 180,E1 -11666.311,E2 -11666.311} C_VEL
LIN {X 0,Y 394.81,Z 501.581,A -85,B 0,C 180,E1 -11668.92,E2 -11668.92} C_VEL
LIN {X 0,Y 396.752,Z 509.183,A -85,B 0,C 180,E1 -11671.427,E2 -11671.427} C_VEL
LIN {X 0,Y 398.295,Z 517.632,A -85,B 0,C 180,E1 -11673.824,E2 -11673.824} C_VEL
LIN {X 0,Y 398.277,Z 519.958,A -85,B 0,C 180,E1 -11674.393,E2 -11674.393} C_VEL
LIN {X 0,Y 395.57,Z 538.632,A -85,B 0,C 180,E1 -11678.436,E2 -11678.436} C_VEL
LIN {X 0,Y 398.641,Z 552.559,A -85,B 0,C 180,E1 -11679.239,E2 -11679.239} C_VEL
LIN {X 0,Y 401.122,Z 568.445,A -85,B 0,C 180,E1 -11679.989,E2 -11679.989} C_VEL
LIN {X 0,Y 397.148,Z 656.733,A -85,B 0,C 180,E1 -11682.426,E2 -11682.426} C_VEL
LIN {X 0,Y 396.427,Z 669.977,A -85,B 0,C 180,E1 -11682.991,E2 -11682.991} C_VEL
LIN {X 0,Y 395.58,Z 682.504,A -85,B 0,C 180,E1 -11683.728,E2 -11683.728} C_VEL
LIN {X 0,Y 394.574,Z 694.546,A -85,B 0,C 180,E1 -11684.636,E2 -11684.636} C_VEL
LIN {X 0,Y 393.539,Z 706.532,A -85,B 0,C 180,E1 -11685.785,E2 -11685.785} C_VEL
LIN {X 0,Y 392.646,Z 715.362,A -85,B 0,C 180,E1 -11686.808,E2 -11686.808} C_VEL
LIN {X 0,Y 391.721,Z 724.53,A -85,B 0,C 180,E1 -11688.093,E2 -11688.093} C_VEL
LIN {X 0,Y 390.964,Z 733.516,A -85,B 0,C 180,E1 -11689.644,E2 -11689.644} C_VEL
LIN {X 0,Y 390.192,Z 740.771,A -85,B 0,C 180,E1 -11691.193,E2 -11691.193} C_VEL
LIN {X 0,Y 389.67,Z 747.59,A -85,B 0,C 180,E1 -11693.074,E2 -11693.074} C_VEL
LIN {X 0,Y 389.093,Z 752.415,A -85,B 0,C 180,E1 -11694.818,E2 -11694.818} C_VEL
LIN {X 0,Y 389.12,Z 754.573,A -85,B 0,C 180,E1 -11695.857,E2 -11695.857} C_VEL
LIN {X 0,Y 389.022,Z 756.273,A -85,B 0,C 180,E1 -11696.893,E2 -11696.893} C_VEL
LIN {X 0,Y 388.85,Z 757.558,A -85,B 0,C 180,E1 -11697.928,E2 -11697.928} C_VEL
LIN {X 0,Y 388.749,Z 758.413,A -85,B 0,C 180,E1 -11698.964,E2 -11698.964} C_VEL
LIN {X 0,Y 388.709,Z 758.799,A -85,B 0,C 180,E1 -11700,E2 -11700} C_VEL
LIN {X 0,Y 388.728,Z 758.768,A -85,B 0,C 180,E1 -11701.036,E2 -11701.036} C_VEL
LIN {X 0,Y 388.736,Z 758.326,A -85,B 0,C 180,E1 -11702.072,E2 -11702.072} C_VEL
LIN {X 0,Y 388.706,Z 757.454,A -85,B 0,C 180,E1 -11703.109,E2 -11703.109} C_VEL
LIN {X 0,Y 388.748,Z 756.114,A -85,B 0,C 180,E1 -11704.147,E2 -11704.147} C_VEL
LIN {X 0,Y 388.868,Z 752.744,A -85,B 0,C 180,E1 -11705.952,E2 -11705.952} C_VEL
LIN {X 0,Y 389.081,Z 747.841,A -85,B 0,C 180,E1 -11707.786,E2 -11707.786} C_VEL
LIN {X 0,Y 389.453,Z 741.238,A -85,B 0,C 180,E1 -11709.609,E2 -11709.609} C_VEL
LIN {X 0,Y 389.855,Z 734.055,A -85,B 0,C 180,E1 -11711.174,E2 -11711.174} C_VEL
LIN {X 0,Y 390.456,Z 726.747,A -85,B 0,C 180,E1 -11712.474,E2 -11712.474} C_VEL
LIN {X 0,Y 391.01,Z 716.81,A -85,B 0,C 180,E1 -11713.927,E2 -11713.927} C_VEL
LIN {X 0,Y 391.793,Z 705.914,A -85,B 0,C 180,E1 -11715.209,E2 -11715.209} C_VEL
LIN {X 0,Y 392.591,Z 695.052,A -85,B 0,C 180,E1 -11716.243,E2 -11716.243} C_VEL
LIN {X 0,Y 393.234,Z 683.063,A -85,B 0,C 180,E1 -11717.151,E2 -11717.151} C_VEL
LIN {X 0,Y 393.899,Z 669.71,A -85,B 0,C 180,E1 -11717.925,E2 -11717.925} C_VEL
LIN {X 0,Y 394.45,Z 656.444,A -85,B 0,C 180,E1 -11718.47,E2 -11718.47} C_VEL
LIN {X 0,Y 394.992,Z 637.097,A -85,B 0,C 180,E1 -11718.96,E2 -11718.96} C_VEL
LIN {X 0,Y 396.597,Z 565.68,A -85,B 0,C 180,E1 -11720.622,E2 -11720.622} C_VEL
LIN {X 0,Y 392.802,Z 539.922,A -85,B 0,C 180,E1 -11721.457,E2 -11721.457} C_VEL
LIN {X 0,Y 394.187,Z 522.132,A -85,B 0,C 180,E1 -11724.864,E2 -11724.864} C_VEL
LIN {X 0,Y 395.147,Z 511.838,A -85,B 0,C 180,E1 -11726.855,E2 -11726.855} C_VEL
LIN {X 0,Y 394.835,Z 508.363,A -85,B 0,C 180,E1 -11727.568,E2 -11727.568} C_VEL
LIN {X 0,Y 391.431,Z 493.071,A -85,B 0,C 180,E1 -11730.895,E2 -11730.895} C_VEL
LIN {X 0,Y 390.045,Z 487.026,A -85,B 0,C 180,E1 -11732.289,E2 -11732.289} C_VEL
LIN {X 0,Y 390.088,Z 487.019,A -85,B 0,C 180,E1 -11735.207,E2 -11735.207} C_VEL
LIN {X 0,Y 390.095,Z 487.016,A -85,B 0,C 180,E1 -11739.092,E2 -11739.092} C_VEL
LIN {X 0,Y 390.045,Z 487.021,A -85,B 0,C 180,E1 -11742.374,E2 -11742.374} C_VEL
LIN {X 0,Y 390.046,Z 487.025,A -85,B 0,C 180,E1 -11745.354,E2 -11745.354} C_VEL
LIN {X 0,Y 390.033,Z 487.023,A -85,B 0,C 180,E1 -11748.187,E2 -11748.187} C_VEL
LIN {X 0,Y 390.089,Z 487.016,A -85,B 0,C 180,E1 -11750.907,E2 -11750.907} C_VEL
LIN {X 0,Y 390.087,Z 487.015,A -85,B 0,C 180,E1 -11754.793,E2 -11754.793} C_VEL
LIN {X 0,Y 390.025,Z 487.023,A -85,B 0,C 180,E1 -11758.496,E2 -11758.496} C_VEL
LIN {X 0,Y 390.119,Z 487.013,A -85,B 0,C 180,E1 -11762.07,E2 -11762.07} C_VEL
LIN {X 0,Y 390.083,Z 487.023,A -85,B 0,C 180,E1 -11765.519,E2 -11765.519} C_VEL
LIN {X 0,Y 390.063,Z 487.019,A -85,B 0,C 180,E1 -11768.878,E2 -11768.878} C_VEL
LIN {X 0,Y 390.13,Z 487.01,A -85,B 0,C 180,E1 -11772.167,E2 -11772.167} C_VEL
LIN {X 0,Y 390.146,Z 487.014,A -85,B 0,C 180,E1 -11775.393,E2 -11775.393} C_VEL
LIN {X 0,Y 390.15,Z 487.007,A -85,B 0,C 180,E1 -11778.571,E2 -11778.571} C_VEL
LIN {X 0,Y 390.346,Z 486.984,A -85,B 0,C 180,E1 -11781.993,E2 -11781.993} C_VEL
LIN {X 0,Y 390.229,Z 486.998,A -85,B 0,C 180,E1 -11784.833,E2 -11784.833} C_VEL
LIN {X 0,Y 390.422,Z 486.975,A -85,B 0,C 180,E1 -11787.937,E2 -11787.937} C_VEL
LIN {X 0,Y 390.552,Z 486.959,A -85,B 0,C 180,E1 -11790,E2 -11790} C_VEL
LIN {X 0,Y 390.317,Z 486.99,A -85,B 0,C 180,E1 -11793.096,E2 -11793.096} C_VEL
LIN {X 0,Y 390.33,Z 486.985,A -85,B 0,C 180,E1 -11796.202,E2 -11796.202} C_VEL
LIN {X 0,Y 390.316,Z 486.987,A -85,B 0,C 180,E1 -11798.282,E2 -11798.282} C_VEL
LIN {X 0,Y 390.143,Z 487.01,A -85,B 0,C 180,E1 -11801.836,E2 -11801.836} C_VEL
LIN {X 0,Y 389.482,Z 487.092,A -85,B 0,C 180,E1 -11802.698,E2 -11802.698} C_VEL
LIN {X 0,Y 386.616,Z 487.448,A -85,B 0,C 180,E1 -11804.1,E2 -11804.1} C_VEL
LIN {X 0,Y 384.189,Z 487.755,A -85,B 0,C 180,E1 -11805.232,E2 -11805.232} C_VEL
LIN {X 0,Y 383.155,Z 487.879,A -85,B 0,C 180,E1 -11806.108,E2 -11806.108} C_VEL
LIN {X 0,Y 383.075,Z 487.889,A -85,B 0,C 180,E1 -11806.405,E2 -11806.405} C_VEL
LIN {X 0,Y 383.062,Z 487.896,A -85,B 0,C 180,E1 -11809.284,E2 -11809.284} C_VEL
LIN {X 0,Y 383.014,Z 487.897,A -85,B 0,C 180,E1 -11812.664,E2 -11812.664} C_VEL
LIN {X 0,Y 383.081,Z 487.888,A -85,B 0,C 180,E1 -11816.123,E2 -11816.123} C_VEL
LIN {X 0,Y 382.993,Z 487.902,A -85,B 0,C 180,E1 -11819.7,E2 -11819.7} C_VEL
LIN {X 0,Y 383.004,Z 487.904,A -85,B 0,C 180,E1 -11823.401,E2 -11823.401} C_VEL
LIN {X 0,Y 383.033,Z 487.894,A -85,B 0,C 180,E1 -11826.165,E2 -11826.165} C_VEL
LIN {X 0,Y 383.011,Z 487.897,A -85,B 0,C 180,E1 -11829.958,E2 -11829.958} C_VEL
LIN {X 0,Y 383.006,Z 487.899,A -85,B 0,C 180,E1 -11832.779,E2 -11832.779} C_VEL
LIN {X 0,Y 382.999,Z 487.9,A -85,B 0,C 180,E1 -11835.79,E2 -11835.79} C_VEL
LIN {X 0,Y 382.989,Z 487.901,A -85,B 0,C 180,E1 -11838.796,E2 -11838.796} C_VEL
LIN {X 0,Y 383.001,Z 487.898,A -85,B 0,C 180,E1 -11842.096,E2 -11842.096} C_VEL
LIN {X 0,Y 383.02,Z 487.902,A -85,B 0,C 180,E1 -11845.332,E2 -11845.332} C_VEL
LIN {X 0,Y 383.004,Z 487.902,A -85,B 0,C 180,E1 -11849.083,E2 -11849.083} C_VEL
LIN {X 0,Y 383.051,Z 487.978,A -85,B 0,C 180,E1 -11849.496,E2 -11849.496} C_VEL
LIN {X 0,Y 386.795,Z 504.651,A -85,B 0,C 180,E1 -11852.607,E2 -11852.607} C_VEL
LIN {X 0,Y 387.894,Z 510.322,A -85,B 0,C 180,E1 -11853.647,E2 -11853.647} C_VEL
LIN {X 0,Y 387.021,Z 526.989,A -85,B 0,C 180,E1 -11856.453,E2 -11856.453} C_VEL
LIN {X 0,Y 386.055,Z 545.09,A -85,B 0,C 180,E1 -11859.486,E2 -11859.486} C_VEL
LIN {X 0,Y 385.934,Z 547.665,A -85,B 0,C 180,E1 -11859.915,E2 -11859.915} C_VEL
LIN {X 0,Y 389.073,Z 569.928,A -85,B 0,C 180,E1 -11860.585,E2 -11860.585} C_VEL
LIN {X 0,Y 387.137,Z 659.385,A -85,B 0,C 180,E1 -11862.672,E2 -11862.672} C_VEL
LIN {X 0,Y 386.594,Z 671.929,A -85,B 0,C 180,E1 -11863.158,E2 -11863.158} C_VEL
LIN {X 0,Y 385.994,Z 684.919,A -85,B 0,C 180,E1 -11863.879,E2 -11863.879} C_VEL
LIN {X 0,Y 385.314,Z 697.387,A -85,B 0,C 180,E1 -11864.8,E2 -11864.8} C_VEL
LIN {X 0,Y 384.713,Z 708.744,A -85,B 0,C 180,E1 -11865.877,E2 -11865.877} C_VEL
LIN {X 0,Y 384.057,Z 718.75,A -85,B 0,C 180,E1 -11867.046,E2 -11867.046} C_VEL
LIN {X 0,Y 383.332,Z 727.945,A -85,B 0,C 180,E1 -11868.365,E2 -11868.365} C_VEL
LIN {X 0,Y 382.738,Z 736.931,A -85,B 0,C 180,E1 -11869.954,E2 -11869.954} C_VEL
LIN {X 0,Y 382.277,Z 744.104,A -85,B 0,C 180,E1 -11871.542,E2 -11871.542} C_VEL
LIN {X 0,Y 382.016,Z 749.97,A -85,B 0,C 180,E1 -11873.185,E2 -11873.185} C_VEL
LIN {X 0,Y 381.83,Z 754.246,A -85,B 0,C 180,E1 -11874.72,E2 -11874.72} C_VEL
LIN {X 0,Y 381.715,Z 756.595,A -85,B 0,C 180,E1 -11875.777,E2 -11875.777} C_VEL
LIN {X 0,Y 381.617,Z 758.428,A -85,B 0,C 180,E1 -11876.833,E2 -11876.833} C_VEL
LIN {X 0,Y 381.619,Z 759.813,A -85,B 0,C 180,E1 -11877.889,E2 -11877.889} C_VEL
LIN {X 0,Y 381.61,Z 760.786,A -85,B 0,C 180,E1 -11878.945,E2 -11878.945} C_VEL
LIN {X 0,Y 381.639,Z 761.287,A -85,B 0,C 180,E1 -11880,E2 -11880} C_VEL
LIN {X 0,Y 381.645,Z 761.358,A -85,B 0,C 180,E1 -11881.055,E2 -11881.055} C_VEL
LIN {X 0,Y 381.701,Z 761.016,A -85,B 0,C 180,E1 -11882.11,E2 -11882.11} C_VEL
LIN {X 0,Y 381.708,Z 760.224,A -85,B 0,C 180,E1 -11883.166,E2 -11883.166} C_VEL
LIN {X 0,Y 381.74,Z 758.981,A -85,B 0,C 180,E1 -11884.223,E2 -11884.223} C_VEL
LIN {X 0,Y 382.105,Z 756.286,A -85,B 0,C 180,E1 -11885.806,E2 -11885.806} C_VEL
LIN {X 0,Y 382.336,Z 752.542,A -85,B 0,C 180,E1 -11887.393,E2 -11887.393} C_VEL
LIN {X 0,Y 382.772,Z 747.619,A -85,B 0,C 180,E1 -11888.979,E2 -11888.979} C_VEL
LIN {X 0,Y 383.37,Z 741.377,A -85,B 0,C 180,E1 -11890.563,E2 -11890.563} C_VEL
LIN {X 0,Y 384.137,Z 733.523,A -85,B 0,C 180,E1 -11892.146,E2 -11892.146} C_VEL
LIN {X 0,Y 385.105,Z 723.756,A -85,B 0,C 180,E1 -11893.724,E2 -11893.724} C_VEL
LIN {X 0,Y 386.24,Z 712.844,A -85,B 0,C 180,E1 -11895.12,E2 -11895.12} C_VEL
LIN {X 0,Y 387.194,Z 702.354,A -85,B 0,C 180,E1 -11896.205,E2 -11896.205} C_VEL
LIN {X 0,Y 387.923,Z 691.361,A -85,B 0,C 180,E1 -11897.122,E2 -11897.122} C_VEL
LIN {X 0,Y 388.956,Z 678.186,A -85,B 0,C 180,E1 -11897.957,E2 -11897.957} C_VEL
LIN {X 0,Y 389.699,Z 664.79,A -85,B 0,C 180,E1 -11898.567,E2 -11898.567} C_VEL
LIN {X 0,Y 390.209,Z 649.889,A -85,B 0,C 180,E1 -11899.019,E2 -11899.019} C_VEL
LIN {X 0,Y 393.27,Z 571.088,A -85,B 0,C 180,E1 -11901.092,E2 -11901.092} C_VEL
LIN {X 0,Y 391.135,Z 557.891,A -85,B 0,C 180,E1 -11901.704,E2 -11901.704} C_VEL
LIN {X 0,Y 389.274,Z 549.53,A -85,B 0,C 180,E1 -11902.176,E2 -11902.176} C_VEL
LIN {X 0,Y 390.922,Z 528.294,A -85,B 0,C 180,E1 -11905.798,E2 -11905.798} C_VEL
LIN {X 0,Y 391.774,Z 518.451,A -85,B 0,C 180,E1 -11907.512,E2 -11907.512} C_VEL
LIN {X 0,Y 390.513,Z 510.859,A -85,B 0,C 180,E1 -11909.072,E2 -11909.072} C_VEL
LIN {X 0,Y 387.959,Z 501.612,A -85,B 0,C 180,E1 -11911.164,E2 -11911.164} C_VEL
LIN {X 0,Y 385.16,Z 493.623,A -85,B 0,C 180,E1 -11913.189,E2 -11913.189} C_VEL
LIN {X 0,Y 383.019,Z 487.902,A -85,B 0,C 180,E1 -11914.828,E2 -11914.828} C_VEL
LIN {X 0,Y 383.002,Z 487.903,A -85,B 0,C 180,E1 -11917.904,E2 -11917.904} C_VEL
LIN {X 0,Y 382.986,Z 487.904,A -85,B 0,C 180,E1 -11921.347,E2 -11921.347} C_VEL
LIN {X 0,Y 382.998,Z 487.902,A -85,B 0,C 180,E1 -11924.303,E2 -11924.303} C_VEL
LIN {X 0,Y 383.041,Z 487.894,A -85,B 0,C 180,E1 -11927.244,E2 -11927.244} C_VEL
LIN {X 0,Y 383.021,Z 487.899,A -85,B 0,C 180,E1 -11930.413,E2 -11930.413} C_VEL
LIN {X 0,Y 383.028,Z 487.898,A -85,B 0,C 180,E1 -11934.045,E2 -11934.045} C_VEL
LIN {X 0,Y 383.039,Z 487.896,A -85,B 0,C 180,E1 -11937.853,E2 -11937.853} C_VEL
LIN {X 0,Y 383.042,Z 487.919,A -85,B 0,C 180,E1 -11938.549,E2 -11938.549} C_VEL
LIN {X 0,Y 387.183,Z 505.1,A -85,B 0,C 180,E1 -11942.069,E2 -11942.069} C_VEL
LIN {X 0,Y 389.119,Z 513.57,A -85,B 0,C 180,E1 -11943.736,E2 -11943.736} C_VEL
LIN {X 0,Y 389.116,Z 516.775,A -85,B 0,C 180,E1 -11944.312,E2 -11944.312} C_VEL
LIN {X 0,Y 388.331,Z 524.324,A -85,B 0,C 180,E1 -11945.598,E2 -11945.598} C_VEL
LIN {X 0,Y 388.751,Z 531.309,A -85,B 0,C 180,E1 -11946.126,E2 -11946.126} C_VEL
LIN {X 0,Y 391.788,Z 552.563,A -85,B 0,C 180,E1 -11946.775,E2 -11946.775} C_VEL
LIN {X 0,Y 389.139,Z 661.964,A -85,B 0,C 180,E1 -11949.207,E2 -11949.207} C_VEL
LIN {X 0,Y 388.453,Z 676.269,A -85,B 0,C 180,E1 -11949.722,E2 -11949.722} C_VEL
LIN {X 0,Y 387.746,Z 690.338,A -85,B 0,C 180,E1 -11950.449,E2 -11950.449} C_VEL
LIN {X 0,Y 386.89,Z 703.269,A -85,B 0,C 180,E1 -11951.327,E2 -11951.327} C_VEL
LIN {X 0,Y 385.964,Z 715.574,A -85,B 0,C 180,E1 -11952.379,E2 -11952.379} C_VEL
LIN {X 0,Y 384.938,Z 727.969,A -85,B 0,C 180,E1 -11953.697,E2 -11953.697} C_VEL
LIN {X 0,Y 384.009,Z 739.086,A -85,B 0,C 180,E1 -11955.154,E2 -11955.154} C_VEL
LIN {X 0,Y 383.268,Z 749.445,A -85,B 0,C 180,E1 -11956.814,E2 -11956.814} C_VEL
LIN {X 0,Y 382.617,Z 758.562,A -85,B 0,C 180,E1 -11958.612,E2 -11958.612} C_VEL
LIN {X 0,Y 382.099,Z 766.094,A -85,B 0,C 180,E1 -11960.472,E2 -11960.472} C_VEL
LIN {X 0,Y 381.839,Z 771.325,A -85,B 0,C 180,E1 -11962.065,E2 -11962.065} C_VEL
LIN {X 0,Y 381.686,Z 776.006,A -85,B 0,C 180,E1 -11963.883,E2 -11963.883} C_VEL
LIN {X 0,Y 381.614,Z 779.571,A -85,B 0,C 180,E1 -11965.775,E2 -11965.775} C_VEL
LIN {X 0,Y 381.614,Z 782.068,A -85,B 0,C 180,E1 -11967.889,E2 -11967.889} C_VEL
LIN {X 0,Y 381.638,Z 783.087,A -85,B 0,C 180,E1 -11970,E2 -11970} C_VEL
LIN {X 0,Y 381.636,Z 783.046,A -85,B 0,C 180,E1 -11971.055,E2 -11971.055} C_VEL
LIN {X 0,Y 381.541,Z 781.866,A -85,B 0,C 180,E1 -11973.168,E2 -11973.168} C_VEL
LIN {X 0,Y 381.612,Z 780.732,A -85,B 0,C 180,E1 -11974.225,E2 -11974.225} C_VEL
LIN {X 0,Y 381.71,Z 777.333,A -85,B 0,C 180,E1 -11976.343,E2 -11976.343} C_VEL
LIN {X 0,Y 381.862,Z 773.708,A -85,B 0,C 180,E1 -11977.934,E2 -11977.934} C_VEL
LIN {X 0,Y 382.193,Z 769.138,A -85,B 0,C 180,E1 -11979.526,E2 -11979.526} C_VEL
LIN {X 0,Y 382.714,Z 762.498,A -85,B 0,C 180,E1 -11981.386,E2 -11981.386} C_VEL
LIN {X 0,Y 383.507,Z 754.216,A -85,B 0,C 180,E1 -11983.242,E2 -11983.242} C_VEL
LIN {X 0,Y 384.386,Z 745.559,A -85,B 0,C 180,E1 -11984.831,E2 -11984.831} C_VEL
LIN {X 0,Y 385.456,Z 735.061,A -85,B 0,C 180,E1 -11986.416,E2 -11986.416} C_VEL
LIN {X 0,Y 386.771,Z 723.334,A -85,B 0,C 180,E1 -11987.857,E2 -11987.857} C_VEL
LIN {X 0,Y 388.06,Z 710.513,A -85,B 0,C 180,E1 -11989.137,E2 -11989.137} C_VEL
LIN {X 0,Y 389.326,Z 697.552,A -85,B 0,C 180,E1 -11990.167,E2 -11990.167} C_VEL
LIN {X 0,Y 390.441,Z 683.508,A -85,B 0,C 180,E1 -11991.031,E2 -11991.031} C_VEL
LIN {X 0,Y 391.432,Z 670.278,A -85,B 0,C 180,E1 -11991.631,E2 -11991.631} C_VEL
LIN {X 0,Y 392.086,Z 655.278,A -85,B 0,C 180,E1 -11992.112,E2 -11992.112} C_VEL
LIN {X 0,Y 394.939,Z 581.288,A -85,B 0,C 180,E1 -11993.921,E2 -11993.921} C_VEL
LIN {X 0,Y 396.089,Z 552.311,A -85,B 0,C 180,E1 -11994.687,E2 -11994.687} C_VEL
LIN {X 0,Y 394.176,Z 539.593,A -85,B 0,C 180,E1 -11995.271,E2 -11995.271} C_VEL
LIN {X 0,Y 391.884,Z 528.497,A -85,B 0,C 180,E1 -11995.9,E2 -11995.9} C_VEL
LIN {X 0,Y 392.831,Z 522.42,A -85,B 0,C 180,E1 -11997.143,E2 -11997.143} C_VEL
LIN {X 0,Y 391.515,Z 515.427,A -85,B 0,C 180,E1 -11998.991,E2 -11998.991} C_VEL
LIN {X 0,Y 389.936,Z 509.055,A -85,B 0,C 180,E1 -12000.909,E2 -12000.909} C_VEL
LIN {X 0,Y 387.768,Z 501.669,A -85,B 0,C 180,E1 -12003.518,E2 -12003.518} C_VEL
LIN {X 0,Y 385.741,Z 495.608,A -85,B 0,C 180,E1 -12006.206,E2 -12006.206} C_VEL
LIN {X 0,Y 384.367,Z 491.761,A -85,B 0,C 180,E1 -12008.439,E2 -12008.439} C_VEL
LIN {X 0,Y 383.084,Z 488.338,A -85,B 0,C 180,E1 -12011.335,E2 -12011.335} C_VEL
LIN {X 0,Y 382.991,Z 487.903,A -85,B 0,C 180,E1 -12012.051,E2 -12012.051} C_VEL
LIN {X 0,Y 382.999,Z 487.902,A -85,B 0,C 180,E1 -12015.697,E2 -12015.697} C_VEL
LIN {X 0,Y 383.013,Z 487.91,A -85,B 0,C 180,E1 -12019.076,E2 -12019.076} C_VEL
LIN {X 0,Y 384.11,Z 490.859,A -85,B 0,C 180,E1 -12021.885,E2 -12021.885} C_VEL
LIN {X 0,Y 385.376,Z 494.755,A -85,B 0,C 180,E1 -12024.298,E2 -12024.298} C_VEL
LIN {X 0,Y 387,Z 499.578,A -85,B 0,C 180,E1 -12026.655,E2 -12026.655} C_VEL
LIN {X 0,Y 388.767,Z 505.661,A -85,B 0,C 180,E1 -12029.076,E2 -12029.076} C_VEL
LIN {X 0,Y 390.761,Z 513.835,A -85,B 0,C 180,E1 -12031.799,E2 -12031.799} C_VEL
LIN {X 0,Y 391.845,Z 520.582,A -85,B 0,C 180,E1 -12033.739,E2 -12033.739} C_VEL
LIN {X 0,Y 391.293,Z 524.894,A -85,B 0,C 180,E1 -12034.75,E2 -12034.75} C_VEL
LIN {X 0,Y 389.157,Z 538.673,A -85,B 0,C 180,E1 -12037.782,E2 -12037.782} C_VEL
LIN {X 0,Y 392.364,Z 552.388,A -85,B 0,C 180,E1 -12038.621,E2 -12038.621} C_VEL
LIN {X 0,Y 395.021,Z 568.99,A -85,B 0,C 180,E1 -12039.459,E2 -12039.459} C_VEL
LIN {X 0,Y 391.808,Z 634.921,A -85,B 0,C 180,E1 -12041.333,E2 -12041.333} C_VEL
LIN {X 0,Y 390.74,Z 657.363,A -85,B 0,C 180,E1 -12041.992,E2 -12041.992} C_VEL
LIN {X 0,Y 389.906,Z 670.961,A -85,B 0,C 180,E1 -12042.603,E2 -12042.603} C_VEL
LIN {X 0,Y 388.953,Z 684.533,A -85,B 0,C 180,E1 -12043.443,E2 -12043.443} C_VEL
LIN {X 0,Y 387.891,Z 696.238,A -85,B 0,C 180,E1 -12044.365,E2 -12044.365} C_VEL
LIN {X 0,Y 386.761,Z 707.898,A -85,B 0,C 180,E1 -12045.531,E2 -12045.531} C_VEL
LIN {X 0,Y 385.823,Z 716.495,A -85,B 0,C 180,E1 -12046.57,E2 -12046.57} C_VEL
LIN {X 0,Y 384.838,Z 725.472,A -85,B 0,C 180,E1 -12047.877,E2 -12047.877} C_VEL
LIN {X 0,Y 384.038,Z 734.336,A -85,B 0,C 180,E1 -12049.455,E2 -12049.455} C_VEL
LIN {X 0,Y 383.231,Z 741.464,A -85,B 0,C 180,E1 -12051.032,E2 -12051.032} C_VEL
LIN {X 0,Y 382.69,Z 747.168,A -85,B 0,C 180,E1 -12052.614,E2 -12052.614} C_VEL
LIN {X 0,Y 382.205,Z 751.651,A -85,B 0,C 180,E1 -12054.195,E2 -12054.195} C_VEL
LIN {X 0,Y 382.045,Z 755.007,A -85,B 0,C 180,E1 -12055.78,E2 -12055.78} C_VEL
LIN {X 0,Y 381.949,Z 756.671,A -85,B 0,C 180,E1 -12056.836,E2 -12056.836} C_VEL
LIN {X 0,Y 381.79,Z 757.922,A -85,B 0,C 180,E1 -12057.89,E2 -12057.89} C_VEL
LIN {X 0,Y 381.682,Z 758.712,A -85,B 0,C 180,E1 -12058.945,E2 -12058.945} C_VEL
LIN {X 0,Y 381.64,Z 759.058,A -85,B 0,C 180,E1 -12060,E2 -12060} C_VEL
LIN {X 0,Y 381.642,Z 758.988,A -85,B 0,C 180,E1 -12061.055,E2 -12061.055} C_VEL
LIN {X 0,Y 381.636,Z 758.503,A -85,B 0,C 180,E1 -12062.111,E2 -12062.111} C_VEL
LIN {X 0,Y 381.613,Z 757.555,A -85,B 0,C 180,E1 -12063.167,E2 -12063.167} C_VEL
LIN {X 0,Y 381.675,Z 756.169,A -85,B 0,C 180,E1 -12064.224,E2 -12064.224} C_VEL
LIN {X 0,Y 381.767,Z 753.056,A -85,B 0,C 180,E1 -12065.902,E2 -12065.902} C_VEL
LIN {X 0,Y 381.944,Z 749.248,A -85,B 0,C 180,E1 -12067.4,E2 -12067.4} C_VEL
LIN {X 0,Y 382.258,Z 743.074,A -85,B 0,C 180,E1 -12069.258,E2 -12069.258} C_VEL
LIN {X 0,Y 382.678,Z 736.258,A -85,B 0,C 180,E1 -12070.85,E2 -12070.85} C_VEL
LIN {X 0,Y 383.36,Z 727.784,A -85,B 0,C 180,E1 -12072.439,E2 -12072.439} C_VEL
LIN {X 0,Y 383.808,Z 719.139,A -85,B 0,C 180,E1 -12073.771,E2 -12073.771} C_VEL
LIN {X 0,Y 384.649,Z 708.619,A -85,B 0,C 180,E1 -12075.092,E2 -12075.092} C_VEL
LIN {X 0,Y 385.478,Z 696.826,A -85,B 0,C 180,E1 -12076.279,E2 -12076.279} C_VEL
LIN {X 0,Y 386.164,Z 685.393,A -85,B 0,C 180,E1 -12077.202,E2 -12077.202} C_VEL
LIN {X 0,Y 386.824,Z 672.745,A -85,B 0,C 180,E1 -12077.991,E2 -12077.991} C_VEL
LIN {X 0,Y 387.434,Z 659.129,A -85,B 0,C 180,E1 -12078.611,E2 -12078.611} C_VEL
LIN {X 0,Y 387.9,Z 644.757,A -85,B 0,C 180,E1 -12079.034,E2 -12079.034} C_VEL
LIN {X 0,Y 389.882,Z 567.242,A -85,B 0,C 180,E1 -12080.874,E2 -12080.874} C_VEL
LIN {X 0,Y 385.889,Z 539.852,A -85,B 0,C 180,E1 -12081.775,E2 -12081.775} C_VEL
LIN {X 0,Y 387.492,Z 520.795,A -85,B 0,C 180,E1 -12085.487,E2 -12085.487} C_VEL
LIN {X 0,Y 388.218,Z 511.68,A -85,B 0,C 180,E1 -12087.288,E2 -12087.288} C_VEL
LIN {X 0,Y 385.815,Z 500.359,A -85,B 0,C 180,E1 -12089.761,E2 -12089.761} C_VEL
LIN {X 0,Y 383.018,Z 487.901,A -85,B 0,C 180,E1 -12092.595,E2 -12092.595} C_VEL
LIN {X 0,Y 383.036,Z 487.895,A -85,B 0,C 180,E1 -12096.165,E2 -12096.165} C_VEL
LIN {X 0,Y 383.012,Z 487.899,A -85,B 0,C 180,E1 -12099.958,E2 -12099.958} C_VEL
LIN {X 0,Y 383.007,Z 487.897,A -85,B 0,C 180,E1 -12102.778,E2 -12102.778} C_VEL
LIN {X 0,Y 382.999,Z 487.903,A -85,B 0,C 180,E1 -12105.789,E2 -12105.789} C_VEL
LIN {X 0,Y 382.989,Z 487.9,A -85,B 0,C 180,E1 -12108.796,E2 -12108.796} C_VEL
LIN {X 0,Y 383,Z 487.899,A -85,B 0,C 180,E1 -12112.096,E2 -12112.096} C_VEL
LIN {X 0,Y 383.019,Z 487.9,A -85,B 0,C 180,E1 -12115.332,E2 -12115.332} C_VEL
LIN {X 0,Y 383.011,Z 487.9,A -85,B 0,C 180,E1 -12117.85,E2 -12117.85} C_VEL
LIN {X 0,Y 383.054,Z 487.896,A -85,B 0,C 180,E1 -12121.723,E2 -12121.723} C_VEL
LIN {X 0,Y 383.054,Z 487.893,A -85,B 0,C 180,E1 -12125.04,E2 -12125.04} C_VEL
LIN {X 0,Y 382.998,Z 487.898,A -85,B 0,C 180,E1 -12128.469,E2 -12128.469} C_VEL
LIN {X 0,Y 383.091,Z 487.89,A -85,B 0,C 180,E1 -12131.828,E2 -12131.828} C_VEL
LIN {X 0,Y 383.112,Z 487.887,A -85,B 0,C 180,E1 -12135.118,E2 -12135.118} C_VEL
LIN {X 0,Y 383.099,Z 487.886,A -85,B 0,C 180,E1 -12138.358,E2 -12138.358} C_VEL
LIN {X 0,Y 383.305,Z 487.862,A -85,B 0,C 180,E1 -12141.933,E2 -12141.933} C_VEL
LIN {X 0,Y 383.201,Z 487.873,A -85,B 0,C 180,E1 -12144.738,E2 -12144.738} C_VEL
LIN {X 0,Y 383.389,Z 487.852,A -85,B 0,C 180,E1 -12147.899,E2 -12147.899} C_VEL
LIN {X 0,Y 383.521,Z 487.834,A -85,B 0,C 180,E1 -12150,E2 -12150} C_VEL
LIN {X 0,Y 383.254,Z 487.87,A -85,B 0,C 180,E1 -12153.154,E2 -12153.154} C_VEL
LIN {X 0,Y 383.287,Z 487.862,A -85,B 0,C 180,E1 -12156.316,E2 -12156.316} C_VEL
LIN {X 0,Y 383.261,Z 487.865,A -85,B 0,C 180,E1 -12158.436,E2 -12158.436} C_VEL
LIN {X 0,Y 383.097,Z 487.888,A -85,B 0,C 180,E1 -12161.836,E2 -12161.836} C_VEL
LIN {X 0,Y 383.112,Z 487.886,A -85,B 0,C 180,E1 -12164.882,E2 -12164.882} C_VEL
LIN {X 0,Y 383.075,Z 487.889,A -85,B 0,C 180,E1 -12166.405,E2 -12166.405} C_VEL
LIN {X 0,Y 382.419,Z 487.976,A -85,B 0,C 180,E1 -12167.282,E2 -12167.282} C_VEL
LIN {X 0,Y 379.562,Z 488.33,A -85,B 0,C 180,E1 -12168.707,E2 -12168.707} C_VEL
LIN {X 0,Y 377.124,Z 488.634,A -85,B 0,C 180,E1 -12169.86,E2 -12169.86} C_VEL
LIN {X 0,Y 376.061,Z 488.764,A -85,B 0,C 180,E1 -12170.751,E2 -12170.751} C_VEL
LIN {X 0,Y 375.966,Z 488.774,A -85,B 0,C 180,E1 -12171.053,E2 -12171.053} C_VEL
LIN {X 0,Y 375.995,Z 488.771,A -85,B 0,C 180,E1 -12174.281,E2 -12174.281} C_VEL
LIN {X 0,Y 376.021,Z 488.768,A -85,B 0,C 180,E1 -12176.652,E2 -12176.652} C_VEL
LIN {X 0,Y 375.966,Z 488.774,A -85,B 0,C 180,E1 -12180.313,E2 -12180.313} C_VEL
LIN {X 0,Y 375.961,Z 488.775,A -85,B 0,C 180,E1 -12184.111,E2 -12184.111} C_VEL
LIN {X 0,Y 375.955,Z 488.777,A -85,B 0,C 180,E1 -12186.741,E2 -12186.741} C_VEL
LIN {X 0,Y 375.991,Z 488.772,A -85,B 0,C 180,E1 -12189.971,E2 -12189.971} C_VEL
LIN {X 0,Y 375.933,Z 488.78,A -85,B 0,C 180,E1 -12193.766,E2 -12193.766} C_VEL
LIN {X 0,Y 375.935,Z 488.78,A -85,B 0,C 180,E1 -12196.811,E2 -12196.811} C_VEL
LIN {X 0,Y 375.964,Z 488.775,A -85,B 0,C 180,E1 -12200.538,E2 -12200.538} C_VEL
LIN {X 0,Y 375.965,Z 488.779,A -85,B 0,C 180,E1 -12203.496,E2 -12203.496} C_VEL
LIN {X 0,Y 375.961,Z 488.778,A -85,B 0,C 180,E1 -12205.889,E2 -12205.889} C_VEL
LIN {X 0,Y 375.987,Z 488.846,A -85,B 0,C 180,E1 -12209.218,E2 -12209.218} C_VEL
LIN {X 0,Y 379.453,Z 504.195,A -85,B 0,C 180,E1 -12212.117,E2 -12212.117} C_VEL
LIN {X 0,Y 380.887,Z 511.233,A -85,B 0,C 180,E1 -12213.424,E2 -12213.424} C_VEL
LIN {X 0,Y 380.527,Z 521.368,A -85,B 0,C 180,E1 -12215.155,E2 -12215.155} C_VEL
LIN {X 0,Y 379.282,Z 542.975,A -85,B 0,C 180,E1 -12218.818,E2 -12218.818} C_VEL
LIN {X 0,Y 379.043,Z 548.123,A -85,B 0,C 180,E1 -12219.642,E2 -12219.642} C_VEL
LIN {X 0,Y 382.183,Z 571.12,A -85,B 0,C 180,E1 -12220.347,E2 -12220.347} C_VEL
LIN {X 0,Y 380.176,Z 659.822,A -85,B 0,C 180,E1 -12222.484,E2 -12222.484} C_VEL
LIN {X 0,Y 379.613,Z 672.232,A -85,B 0,C 180,E1 -12222.978,E2 -12222.978} C_VEL
LIN {X 0,Y 379.005,Z 685.181,A -85,B 0,C 180,E1 -12223.712,E2 -12223.712} C_VEL
LIN {X 0,Y 378.307,Z 697.625,A -85,B 0,C 180,E1 -12224.649,E2 -12224.649} C_VEL
LIN {X 0,Y 377.715,Z 708.301,A -85,B 0,C 180,E1 -12225.674,E2 -12225.674} C_VEL
LIN {X 0,Y 377.013,Z 718.986,A -85,B 0,C 180,E1 -12226.937,E2 -12226.937} C_VEL
LIN {X 0,Y 376.233,Z 729.006,A -85,B 0,C 180,E1 -12228.416,E2 -12228.416} C_VEL
LIN {X 0,Y 375.621,Z 737.849,A -85,B 0,C 180,E1 -12230.034,E2 -12230.034} C_VEL
LIN {X 0,Y 375.144,Z 744.867,A -85,B 0,C 180,E1 -12231.652,E2 -12231.652} C_VEL
LIN {X 0,Y 374.865,Z 751.307,A -85,B 0,C 180,E1 -12233.541,E2 -12233.541} C_VEL
LIN {X 0,Y 374.711,Z 755.45,A -85,B 0,C 180,E1 -12235.158,E2 -12235.158} C_VEL
LIN {X 0,Y 374.53,Z 758.477,A -85,B 0,C 180,E1 -12236.773,E2 -12236.773} C_VEL
LIN {X 0,Y 374.519,Z 759.902,A -85,B 0,C 180,E1 -12237.849,E2 -12237.849} C_VEL
LIN {X 0,Y 374.511,Z 760.911,A -85,B 0,C 180,E1 -12238.925,E2 -12238.925} C_VEL
LIN {X 0,Y 374.554,Z 761.476,A -85,B 0,C 180,E1 -12240,E2 -12240} C_VEL
LIN {X 0,Y 374.563,Z 761.58,A -85,B 0,C 180,E1 -12241.075,E2 -12241.075} C_VEL
LIN {X 0,Y 374.606,Z 761.272,A -85,B 0,C 180,E1 -12242.15,E2 -12242.15} C_VEL
LIN {X 0,Y 374.618,Z 760.545,A -85,B 0,C 180,E1 -12243.226,E2 -12243.226} C_VEL
LIN {X 0,Y 374.674,Z 759.342,A -85,B 0,C 180,E1 -12244.303,E2 -12244.303} C_VEL
LIN {X 0,Y 375.069,Z 756.715,A -85,B 0,C 180,E1 -12245.915,E2 -12245.915} C_VEL
LIN {X 0,Y 375.31,Z 753.031,A -85,B 0,C 180,E1 -12247.532,E2 -12247.532} C_VEL
LIN {X 0,Y 375.772,Z 748.163,A -85,B 0,C 180,E1 -12249.147,E2 -12249.147} C_VEL
LIN {X 0,Y 376.419,Z 741.99,A -85,B 0,C 180,E1 -12250.761,E2 -12250.761} C_VEL
LIN {X 0,Y 377.263,Z 734.293,A -85,B 0,C 180,E1 -12252.371,E2 -12252.371} C_VEL
LIN {X 0,Y 378.119,Z 726.432,A -85,B 0,C 180,E1 -12253.708,E2 -12253.708} C_VEL
LIN {X 0,Y 379.137,Z 716.881,A -85,B 0,C 180,E1 -12255.041,E2 -12255.041} C_VEL
LIN {X 0,Y 380.208,Z 706.3,A -85,B 0,C 180,E1 -12256.235,E2 -12256.235} C_VEL
LIN {X 0,Y 381.289,Z 692.968,A -85,B 0,C 180,E1 -12257.429,E2 -12257.429} C_VEL
LIN {X 0,Y 382.415,Z 679.204,A -85,B 0,C 180,E1 -12258.344,E2 -12258.344} C_VEL
LIN {X 0,Y 383.199,Z 666.439,A -85,B 0,C 180,E1 -12258.964,E2 -12258.964} C_VEL
LIN {X 0,Y 383.804,Z 652.429,A -85,B 0,C 180,E1 -12259.419,E2 -12259.419} C_VEL
LIN {X 0,Y 386.783,Z 582.394,A -85,B 0,C 180,E1 -12261.31,E2 -12261.31} C_VEL
LIN {X 0,Y 387.07,Z 571.491,A -85,B 0,C 180,E1 -12261.636,E2 -12261.636} C_VEL
LIN {X 0,Y 385.023,Z 559.146,A -85,B 0,C 180,E1 -12262.239,E2 -12262.239} C_VEL
LIN {X 0,Y 382.978,Z 549.817,A -85,B 0,C 180,E1 -12262.798,E2 -12262.798} C_VEL
LIN {X 0,Y 384.82,Z 528.473,A -85,B 0,C 180,E1 -12266.505,E2 -12266.505} C_VEL
LIN {X 0,Y 385.462,Z 521.577,A -85,B 0,C 180,E1 -12267.706,E2 -12267.706} C_VEL
LIN {X 0,Y 384.885,Z 516.481,A -85,B 0,C 180,E1 -12268.779,E2 -12268.779} C_VEL
LIN {X 0,Y 383.15,Z 509.122,A -85,B 0,C 180,E1 -12270.446,E2 -12270.446} C_VEL
LIN {X 0,Y 380.38,Z 500.3,A -85,B 0,C 180,E1 -12272.641,E2 -12272.641} C_VEL
LIN {X 0,Y 377.329,Z 492.131,A -85,B 0,C 180,E1 -12274.962,E2 -12274.962} C_VEL
LIN {X 0,Y 375.992,Z 488.775,A -85,B 0,C 180,E1 -12276.072,E2 -12276.072} C_VEL
LIN {X 0,Y 375.99,Z 488.775,A -85,B 0,C 180,E1 -12279.971,E2 -12279.971} C_VEL
LIN {X 0,Y 375.931,Z 488.779,A -85,B 0,C 180,E1 -12283.766,E2 -12283.766} C_VEL
LIN {X 0,Y 375.962,Z 488.777,A -85,B 0,C 180,E1 -12287.704,E2 -12287.704} C_VEL
LIN {X 0,Y 375.968,Z 488.777,A -85,B 0,C 180,E1 -12290.538,E2 -12290.538} C_VEL
LIN {X 0,Y 375.967,Z 488.778,A -85,B 0,C 180,E1 -12293.495,E2 -12293.495} C_VEL
LIN {X 0,Y 375.965,Z 488.777,A -85,B 0,C 180,E1 -12295.889,E2 -12295.889} C_VEL
LIN {X 0,Y 376.017,Z 488.858,A -85,B 0,C 180,E1 -12298.207,E2 -12298.207} C_VEL
LIN {X 0,Y 379.872,Z 504.824,A -85,B 0,C 180,E1 -12301.55,E2 -12301.55} C_VEL
LIN {X 0,Y 382.337,Z 516.209,A -85,B 0,C 180,E1 -12303.822,E2 -12303.822} C_VEL
LIN {X 0,Y 382.059,Z 519.512,A -85,B 0,C 180,E1 -12304.398,E2 -12304.398} C_VEL
LIN {X 0,Y 382.959,Z 531.687,A -85,B 0,C 180,E1 -12305.468,E2 -12305.468} C_VEL
LIN {X 0,Y 383.165,Z 540.219,A -85,B 0,C 180,E1 -12306.073,E2 -12306.073} C_VEL
LIN {X 0,Y 384.961,Z 552.423,A -85,B 0,C 180,E1 -12306.456,E2 -12306.456} C_VEL
LIN {X 0,Y 382.211,Z 662.738,A -85,B 0,C 180,E1 -12308.988,E2 -12308.988} C_VEL
LIN {X 0,Y 381.461,Z 677.479,A -85,B 0,C 180,E1 -12309.546,E2 -12309.546} C_VEL
LIN {X 0,Y 380.773,Z 690.996,A -85,B 0,C 180,E1 -12310.274,E2 -12310.274} C_VEL
LIN {X 0,Y 379.867,Z 704.778,A -85,B 0,C 180,E1 -12311.249,E2 -12311.249} C_VEL
LIN {X 0,Y 378.894,Z 716.718,A -85,B 0,C 180,E1 -12312.318,E2 -12312.318} C_VEL
LIN {X 0,Y 377.84,Z 728.856,A -85,B 0,C 180,E1 -12313.66,E2 -12313.66} C_VEL
LIN {X 0,Y 376.897,Z 739.806,A -85,B 0,C 180,E1 -12315.144,E2 -12315.144} C_VEL
LIN {X 0,Y 376.191,Z 750.053,A -85,B 0,C 180,E1 -12316.84,E2 -12316.84} C_VEL
LIN {X 0,Y 375.502,Z 758.963,A -85,B 0,C 180,E1 -12318.666,E2 -12318.666} C_VEL
LIN {X 0,Y 375.05,Z 765.45,A -85,B 0,C 180,E1 -12320.291,E2 -12320.291} C_VEL
LIN {X 0,Y 374.787,Z 770.76,A -85,B 0,C 180,E1 -12321.915,E2 -12321.915} C_VEL
LIN {X 0,Y 374.611,Z 775.804,A -85,B 0,C 180,E1 -12323.893,E2 -12323.893} C_VEL
LIN {X 0,Y 374.54,Z 779.175,A -85,B 0,C 180,E1 -12325.696,E2 -12325.696} C_VEL
LIN {X 0,Y 374.513,Z 781.754,A -85,B 0,C 180,E1 -12327.849,E2 -12327.849} C_VEL
LIN {X 0,Y 374.555,Z 782.478,A -85,B 0,C 180,E1 -12328.925,E2 -12328.925} C_VEL
LIN {X 0,Y 374.537,Z 782.819,A -85,B 0,C 180,E1 -12331.075,E2 -12331.075} C_VEL
LIN {X 0,Y 374.456,Z 781.693,A -85,B 0,C 180,E1 -12333.228,E2 -12333.228} C_VEL
LIN {X 0,Y 374.516,Z 780.583,A -85,B 0,C 180,E1 -12334.305,E2 -12334.305} C_VEL
LIN {X 0,Y 374.63,Z 777.244,A -85,B 0,C 180,E1 -12336.463,E2 -12336.463} C_VEL
LIN {X 0,Y 374.805,Z 773.664,A -85,B 0,C 180,E1 -12338.085,E2 -12338.085} C_VEL
LIN {X 0,Y 375.137,Z 769.149,A -85,B 0,C 180,E1 -12339.707,E2 -12339.707} C_VEL
LIN {X 0,Y 375.737,Z 762.569,A -85,B 0,C 180,E1 -12341.6,E2 -12341.6} C_VEL
LIN {X 0,Y 376.552,Z 754.473,A -85,B 0,C 180,E1 -12343.468,E2 -12343.468} C_VEL
LIN {X 0,Y 377.509,Z 745.784,A -85,B 0,C 180,E1 -12345.108,E2 -12345.108} C_VEL
LIN {X 0,Y 378.661,Z 735.438,A -85,B 0,C 180,E1 -12346.719,E2 -12346.719} C_VEL
LIN {X 0,Y 380.032,Z 723.849,A -85,B 0,C 180,E1 -12348.184,E2 -12348.184} C_VEL
LIN {X 0,Y 381.391,Z 711.242,A -85,B 0,C 180,E1 -12349.482,E2 -12349.482} C_VEL
LIN {X 0,Y 382.771,Z 698.333,A -85,B 0,C 180,E1 -12350.544,E2 -12350.544} C_VEL
LIN {X 0,Y 383.928,Z 685.018,A -85,B 0,C 180,E1 -12351.406,E2 -12351.406} C_VEL
LIN {X 0,Y 384.933,Z 672.486,A -85,B 0,C 180,E1 -12352.015,E2 -12352.015} C_VEL
LIN {X 0,Y 385.757,Z 657.611,A -85,B 0,C 180,E1 -12352.53,E2 -12352.53} C_VEL
LIN {X 0,Y 389.083,Z 577.424,A -85,B 0,C 180,E1 -12354.578,E2 -12354.578} C_VEL
LIN {X 0,Y 390.144,Z 553.026,A -85,B 0,C 180,E1 -12355.247,E2 -12355.247} C_VEL
LIN {X 0,Y 387.927,Z 539.009,A -85,B 0,C 180,E1 -12355.942,E2 -12355.942} C_VEL
LIN {X 0,Y 385.752,Z 528.83,A -85,B 0,C 180,E1 -12356.559,E2 -12356.559} C_VEL
LIN {X 0,Y 386.406,Z 525.141,A -85,B 0,C 180,E1 -12357.339,E2 -12357.339} C_VEL
LIN {X 0,Y 385.149,Z 518.222,A -85,B 0,C 180,E1 -12359.227,E2 -12359.227} C_VEL
LIN {X 0,Y 383.332,Z 511.087,A -85,B 0,C 180,E1 -12361.476,E2 -12361.476} C_VEL
LIN {X 0,Y 381.468,Z 504.381,A -85,B 0,C 180,E1 -12363.998,E2 -12363.998} C_VEL
LIN {X 0,Y 379.817,Z 499.463,A -85,B 0,C 180,E1 -12366.308,E2 -12366.308} C_VEL
LIN {X 0,Y 378.957,Z 496.968,A -85,B 0,C 180,E1 -12367.735,E2 -12367.735} C_VEL
LIN {X 0,Y 377.666,Z 493.626,A -85,B 0,C 180,E1 -12370.273,E2 -12370.273} C_VEL
LIN {X 0,Y 377.144,Z 491.913,A -85,B 0,C 180,E1 -12372.133,E2 -12372.133} C_VEL
LIN {X 0,Y 376.553,Z 490.932,A -85,B 0,C 180,E1 -12374.827,E2 -12374.827} C_VEL
LIN {X 0,Y 376.641,Z 491.043,A -85,B 0,C 180,E1 -12376.697,E2 -12376.697} C_VEL
LIN {X 0,Y 377.315,Z 492.28,A -85,B 0,C 180,E1 -12379.313,E2 -12379.313} C_VEL
LIN {X 0,Y 378.389,Z 495.39,A -85,B 0,C 180,E1 -12382.199,E2 -12382.199} C_VEL
LIN {X 0,Y 379.913,Z 499.986,A -85,B 0,C 180,E1 -12385.008,E2 -12385.008} C_VEL
LIN {X 0,Y 381.259,Z 504.369,A -85,B 0,C 180,E1 -12387.078,E2 -12387.078} C_VEL
LIN {X 0,Y 383.006,Z 510.719,A -85,B 0,C 180,E1 -12389.591,E2 -12389.591} C_VEL
LIN {X 0,Y 384.584,Z 517.709,A -85,B 0,C 180,E1 -12391.929,E2 -12391.929} C_VEL
LIN {X 0,Y 385.397,Z 523.729,A -85,B 0,C 180,E1 -12393.682,E2 -12393.682} C_VEL
LIN {X 0,Y 382.884,Z 538.553,A -85,B 0,C 180,E1 -12397.064,E2 -12397.064} C_VEL
LIN {X 0,Y 386.444,Z 553.761,A -85,B 0,C 180,E1 -12398.05,E2 -12398.05} C_VEL
LIN {X 0,Y 388.937,Z 569.555,A -85,B 0,C 180,E1 -12398.895,E2 -12398.895} C_VEL
LIN {X 0,Y 386.111,Z 624.355,A -85,B 0,C 180,E1 -12400.529,E2 -12400.529} C_VEL
LIN {X 0,Y 384.428,Z 657.46,A -85,B 0,C 180,E1 -12401.514,E2 -12401.514} C_VEL
LIN {X 0,Y 383.56,Z 670.926,A -85,B 0,C 180,E1 -12402.127,E2 -12402.127} C_VEL
LIN {X 0,Y 382.556,Z 683.472,A -85,B 0,C 180,E1 -12402.906,E2 -12402.906} C_VEL
LIN {X 0,Y 381.32,Z 696.532,A -85,B 0,C 180,E1 -12403.951,E2 -12403.951} C_VEL
LIN {X 0,Y 379.99,Z 709.277,A -85,B 0,C 180,E1 -12405.267,E2 -12405.267} C_VEL
LIN {X 0,Y 379.019,Z 717.703,A -85,B 0,C 180,E1 -12406.325,E2 -12406.325} C_VEL
LIN {X 0,Y 378.001,Z 726.544,A -85,B 0,C 180,E1 -12407.654,E2 -12407.654} C_VEL
LIN {X 0,Y 377.117,Z 735.195,A -85,B 0,C 180,E1 -12409.259,E2 -12409.259} C_VEL
LIN {X 0,Y 376.277,Z 742.174,A -85,B 0,C 180,E1 -12410.865,E2 -12410.865} C_VEL
LIN {X 0,Y 375.67,Z 747.98,A -85,B 0,C 180,E1 -12412.536,E2 -12412.536} C_VEL
LIN {X 0,Y 375.177,Z 752.2,A -85,B 0,C 180,E1 -12414.086,E2 -12414.086} C_VEL
LIN {X 0,Y 374.973,Z 755.48,A -85,B 0,C 180,E1 -12415.7,E2 -12415.7} C_VEL
LIN {X 0,Y 374.88,Z 757.101,A -85,B 0,C 180,E1 -12416.776,E2 -12416.776} C_VEL
LIN {X 0,Y 374.732,Z 758.293,A -85,B 0,C 180,E1 -12417.85,E2 -12417.85} C_VEL
LIN {X 0,Y 374.618,Z 759.013,A -85,B 0,C 180,E1 -12418.925,E2 -12418.925} C_VEL
LIN {X 0,Y 374.574,Z 759.316,A -85,B 0,C 180,E1 -12420,E2 -12420} C_VEL
LIN {X 0,Y 374.559,Z 759.206,A -85,B 0,C 180,E1 -12421.075,E2 -12421.075} C_VEL
LIN {X 0,Y 374.536,Z 758.662,A -85,B 0,C 180,E1 -12422.151,E2 -12422.151} C_VEL
LIN {X 0,Y 374.524,Z 757.652,A -85,B 0,C 180,E1 -12423.227,E2 -12423.227} C_VEL
LIN {X 0,Y 374.605,Z 756.217,A -85,B 0,C 180,E1 -12424.304,E2 -12424.304} C_VEL
LIN {X 0,Y 374.712,Z 752.493,A -85,B 0,C 180,E1 -12426.249,E2 -12426.249} C_VEL
LIN {X 0,Y 374.944,Z 747.469,A -85,B 0,C 180,E1 -12428.081,E2 -12428.081} C_VEL
LIN {X 0,Y 375.354,Z 740.624,A -85,B 0,C 180,E1 -12429.974,E2 -12429.974} C_VEL
LIN {X 0,Y 375.858,Z 733.151,A -85,B 0,C 180,E1 -12431.596,E2 -12431.596} C_VEL
LIN {X 0,Y 376.433,Z 725.546,A -85,B 0,C 180,E1 -12432.946,E2 -12432.946} C_VEL
LIN {X 0,Y 377.111,Z 715.345,A -85,B 0,C 180,E1 -12434.433,E2 -12434.433} C_VEL
LIN {X 0,Y 377.861,Z 705.13,A -85,B 0,C 180,E1 -12435.646,E2 -12435.646} C_VEL
LIN {X 0,Y 378.731,Z 693.951,A -85,B 0,C 180,E1 -12436.716,E2 -12436.716} C_VEL
LIN {X 0,Y 379.433,Z 681.654,A -85,B 0,C 180,E1 -12437.656,E2 -12437.656} C_VEL
LIN {X 0,Y 380.053,Z 669.155,A -85,B 0,C 180,E1 -12438.392,E2 -12438.392} C_VEL
LIN {X 0,Y 380.658,Z 655.643,A -85,B 0,C 180,E1 -12438.955,E2 -12438.955} C_VEL
LIN {X 0,Y 381.358,Z 630.994,A -85,B 0,C 180,E1 -12439.597,E2 -12439.597} C_VEL
LIN {X 0,Y 382.991,Z 567.683,A -85,B 0,C 180,E1 -12441.161,E2 -12441.161} C_VEL
LIN {X 0,Y 378.963,Z 539.814,A -85,B 0,C 180,E1 -12442.086,E2 -12442.086} C_VEL
LIN {X 0,Y 380.594,Z 521.484,A -85,B 0,C 180,E1 -12445.718,E2 -12445.718} C_VEL
LIN {X 0,Y 381.299,Z 512.933,A -85,B 0,C 180,E1 -12447.438,E2 -12447.438} C_VEL
LIN {X 0,Y 378.427,Z 499.747,A -85,B 0,C 180,E1 -12450.378,E2 -12450.378} C_VEL
LIN {X 0,Y 375.974,Z 488.779,A -85,B 0,C 180,E1 -12452.946,E2 -12452.946} C_VEL
LIN {X 0,Y 375.967,Z 488.775,A -85,B 0,C 180,E1 -12456.505,E2 -12456.505} C_VEL
LIN {X 0,Y 375.992,Z 488.774,A -85,B 0,C 180,E1 -12459.971,E2 -12459.971} C_VEL
LIN {X 0,Y 375.932,Z 488.783,A -85,B 0,C 180,E1 -12463.766,E2 -12463.766} C_VEL
LIN {X 0,Y 375.935,Z 488.778,A -85,B 0,C 180,E1 -12466.81,E2 -12466.81} C_VEL
LIN {X 0,Y 375.962,Z 488.775,A -85,B 0,C 180,E1 -12470.537,E2 -12470.537} C_VEL
LIN {X 0,Y 375.965,Z 488.78,A -85,B 0,C 180,E1 -12473.495,E2 -12473.495} C_VEL
LIN {X 0,Y 375.961,Z 488.778,A -85,B 0,C 180,E1 -12475.888,E2 -12475.888} C_VEL
LIN {X 0,Y 375.966,Z 488.779,A -85,B 0,C 180,E1 -12479.687,E2 -12479.687} C_VEL
LIN {X 0,Y 375.997,Z 488.771,A -85,B 0,C 180,E1 -12482.141,E2 -12482.141} C_VEL
LIN {X 0,Y 376.008,Z 488.769,A -85,B 0,C 180,E1 -12484.539,E2 -12484.539} C_VEL
LIN {X 0,Y 375.967,Z 488.776,A -85,B 0,C 180,E1 -12488.046,E2 -12488.046} C_VEL
LIN {X 0,Y 376.026,Z 488.773,A -85,B 0,C 180,E1 -12491.474,E2 -12491.474} C_VEL
LIN {X 0,Y 376.06,Z 488.763,A -85,B 0,C 180,E1 -12494.833,E2 -12494.833} C_VEL
LIN {X 0,Y 376.052,Z 488.764,A -85,B 0,C 180,E1 -12498.137,E2 -12498.137} C_VEL
LIN {X 0,Y 376.259,Z 488.74,A -85,B 0,C 180,E1 -12501.877,E2 -12501.877} C_VEL
LIN {X 0,Y 376.174,Z 488.749,A -85,B 0,C 180,E1 -12504.64,E2 -12504.64} C_VEL
LIN {X 0,Y 376.356,Z 488.728,A -85,B 0,C 180,E1 -12507.86,E2 -12507.86} C_VEL
LIN {X 0,Y 376.491,Z 488.71,A -85,B 0,C 180,E1 -12510,E2 -12510} C_VEL
LIN {X 0,Y 376.192,Z 488.75,A -85,B 0,C 180,E1 -12513.213,E2 -12513.213} C_VEL
LIN {X 0,Y 376.247,Z 488.739,A -85,B 0,C 180,E1 -12516.435,E2 -12516.435} C_VEL
LIN {X 0,Y 376.207,Z 488.744,A -85,B 0,C 180,E1 -12518.595,E2 -12518.595} C_VEL
LIN {X 0,Y 376.052,Z 488.766,A -85,B 0,C 180,E1 -12521.863,E2 -12521.863} C_VEL
LIN {X 0,Y 376.06,Z 488.767,A -85,B 0,C 180,E1 -12525.167,E2 -12525.167} C_VEL
LIN {X 0,Y 376.01,Z 488.769,A -85,B 0,C 180,E1 -12528.527,E2 -12528.527} C_VEL
LIN {X 0,Y 375.966,Z 488.774,A -85,B 0,C 180,E1 -12531.053,E2 -12531.053} C_VEL
LIN {X 0,Y 375.271,Z 488.863,A -85,B 0,C 180,E1 -12531.948,E2 -12531.948} C_VEL
LIN {X 0,Y 372.404,Z 489.225,A -85,B 0,C 180,E1 -12533.402,E2 -12533.402} C_VEL
LIN {X 0,Y 370.021,Z 489.516,A -85,B 0,C 180,E1 -12534.578,E2 -12534.578} C_VEL
LIN {X 0,Y 369.042,Z 489.642,A -85,B 0,C 180,E1 -12535.488,E2 -12535.488} C_VEL
LIN {X 0,Y 368.984,Z 489.644,A -85,B 0,C 180,E1 -12535.796,E2 -12535.796} C_VEL
LIN {X 0,Y 368.948,Z 489.65,A -85,B 0,C 180,E1 -12538.808,E2 -12538.808} C_VEL
LIN {X 0,Y 368.899,Z 489.655,A -85,B 0,C 180,E1 -12542.238,E2 -12542.238} C_VEL
LIN {X 0,Y 368.93,Z 489.654,A -85,B 0,C 180,E1 -12545.002,E2 -12545.002} C_VEL
LIN {X 0,Y 368.91,Z 489.654,A -85,B 0,C 180,E1 -12548.641,E2 -12548.641} C_VEL
LIN {X 0,Y 368.883,Z 489.657,A -85,B 0,C 180,E1 -12552.01,E2 -12552.01} C_VEL
LIN {X 0,Y 368.928,Z 489.656,A -85,B 0,C 180,E1 -12555.183,E2 -12555.183} C_VEL
LIN {X 0,Y 368.884,Z 489.657,A -85,B 0,C 180,E1 -12558.178,E2 -12558.178} C_VEL
LIN {X 0,Y 368.91,Z 489.659,A -85,B 0,C 180,E1 -12561.36,E2 -12561.36} C_VEL
LIN {X 0,Y 368.938,Z 489.655,A -85,B 0,C 180,E1 -12565.147,E2 -12565.147} C_VEL
LIN {X 0,Y 368.941,Z 489.753,A -85,B 0,C 180,E1 -12568.924,E2 -12568.924} C_VEL
LIN {X 0,Y 372.69,Z 506.291,A -85,B 0,C 180,E1 -12572.095,E2 -12572.095} C_VEL
LIN {X 0,Y 374.052,Z 513.845,A -85,B 0,C 180,E1 -12573.498,E2 -12573.498} C_VEL
LIN {X 0,Y 373.102,Z 530.731,A -85,B 0,C 180,E1 -12576.404,E2 -12576.404} C_VEL
LIN {X 0,Y 372.1,Z 548.13,A -85,B 0,C 180,E1 -12579.348,E2 -12579.348} C_VEL
LIN {X 0,Y 375.31,Z 571.479,A -85,B 0,C 180,E1 -12580.09,E2 -12580.09} C_VEL
LIN {X 0,Y 373.212,Z 659.144,A -85,B 0,C 180,E1 -12582.252,E2 -12582.252} C_VEL
LIN {X 0,Y 372.639,Z 672.537,A -85,B 0,C 180,E1 -12582.79,E2 -12582.79} C_VEL
LIN {X 0,Y 372.016,Z 685.44,A -85,B 0,C 180,E1 -12583.538,E2 -12583.538} C_VEL
LIN {X 0,Y 371.301,Z 697.862,A -85,B 0,C 180,E1 -12584.493,E2 -12584.493} C_VEL
LIN {X 0,Y 370.702,Z 708.56,A -85,B 0,C 180,E1 -12585.54,E2 -12585.54} C_VEL
LIN {X 0,Y 369.974,Z 719.222,A -85,B 0,C 180,E1 -12586.824,E2 -12586.824} C_VEL
LIN {X 0,Y 369.215,Z 728.424,A -85,B 0,C 180,E1 -12588.192,E2 -12588.192} C_VEL
LIN {X 0,Y 368.588,Z 737.428,A -85,B 0,C 180,E1 -12589.841,E2 -12589.841} C_VEL
LIN {X 0,Y 368.107,Z 744.6,A -85,B 0,C 180,E1 -12591.491,E2 -12591.491} C_VEL
LIN {X 0,Y 367.801,Z 751.137,A -85,B 0,C 180,E1 -12593.417,E2 -12593.417} C_VEL
LIN {X 0,Y 367.628,Z 755.385,A -85,B 0,C 180,E1 -12595.065,E2 -12595.065} C_VEL
LIN {X 0,Y 367.447,Z 758.5,A -85,B 0,C 180,E1 -12596.711,E2 -12596.711} C_VEL
LIN {X 0,Y 367.419,Z 759.973,A -85,B 0,C 180,E1 -12597.808,E2 -12597.808} C_VEL
LIN {X 0,Y 367.412,Z 761.02,A -85,B 0,C 180,E1 -12598.904,E2 -12598.904} C_VEL
LIN {X 0,Y 367.457,Z 761.652,A -85,B 0,C 180,E1 -12600,E2 -12600} C_VEL
LIN {X 0,Y 367.467,Z 761.807,A -85,B 0,C 180,E1 -12601.096,E2 -12601.096} C_VEL
LIN {X 0,Y 367.511,Z 761.538,A -85,B 0,C 180,E1 -12602.192,E2 -12602.192} C_VEL
LIN {X 0,Y 367.529,Z 760.859,A -85,B 0,C 180,E1 -12603.289,E2 -12603.289} C_VEL
LIN {X 0,Y 367.612,Z 759.71,A -85,B 0,C 180,E1 -12604.386,E2 -12604.386} C_VEL
LIN {X 0,Y 368.035,Z 757.143,A -85,B 0,C 180,E1 -12606.029,E2 -12606.029} C_VEL
LIN {X 0,Y 368.29,Z 753.531,A -85,B 0,C 180,E1 -12607.677,E2 -12607.677} C_VEL
LIN {X 0,Y 368.783,Z 748.767,A -85,B 0,C 180,E1 -12609.322,E2 -12609.322} C_VEL
LIN {X 0,Y 369.476,Z 742.704,A -85,B 0,C 180,E1 -12610.965,E2 -12610.965} C_VEL
LIN {X 0,Y 370.381,Z 735.13,A -85,B 0,C 180,E1 -12612.604,E2 -12612.604} C_VEL
LIN {X 0,Y 371.446,Z 725.619,A -85,B 0,C 180,E1 -12614.239,E2 -12614.239} C_VEL
LIN {X 0,Y 372.555,Z 716.531,A -85,B 0,C 180,E1 -12615.509,E2 -12615.509} C_VEL
LIN {X 0,Y 373.629,Z 706.394,A -85,B 0,C 180,E1 -12616.67,E2 -12616.67} C_VEL
LIN {X 0,Y 374.656,Z 694.742,A -85,B 0,C 180,E1 -12617.748,E2 -12617.748} C_VEL
LIN {X 0,Y 375.739,Z 682.627,A -85,B 0,C 180,E1 -12618.611,E2 -12618.611} C_VEL
LIN {X 0,Y 376.734,Z 668.143,A -85,B 0,C 180,E1 -12619.373,E2 -12619.373} C_VEL
LIN {X 0,Y 377.47,Z 652.726,A -85,B 0,C 180,E1 -12619.9,E2 -12619.9} C_VEL
LIN {X 0,Y 381.147,Z 573.934,A -85,B 0,C 180,E1 -12622.117,E2 -12622.117} C_VEL
LIN {X 0,Y 379.491,Z 562.61,A -85,B 0,C 180,E1 -12622.687,E2 -12622.687} C_VEL
LIN {X 0,Y 376.744,Z 550.056,A -85,B 0,C 180,E1 -12623.466,E2 -12623.466} C_VEL
LIN {X 0,Y 378.869,Z 528.296,A -85,B 0,C 180,E1 -12627.316,E2 -12627.316} C_VEL
LIN {X 0,Y 379.257,Z 523.511,A -85,B 0,C 180,E1 -12628.199,E2 -12628.199} C_VEL
LIN {X 0,Y 378.077,Z 516.219,A -85,B 0,C 180,E1 -12629.818,E2 -12629.818} C_VEL
LIN {X 0,Y 375.739,Z 507.592,A -85,B 0,C 180,E1 -12631.95,E2 -12631.95} C_VEL
LIN {X 0,Y 372.615,Z 498.698,A -85,B 0,C 180,E1 -12634.461,E2 -12634.461} C_VEL
LIN {X 0,Y 370.711,Z 493.94,A -85,B 0,C 180,E1 -12635.994,E2 -12635.994} C_VEL
LIN {X 0,Y 368.993,Z 490.261,A -85,B 0,C 180,E1 -12637.352,E2 -12637.352} C_VEL
LIN {X 0,Y 368.906,Z 489.657,A -85,B 0,C 180,E1 -12637.563,E2 -12637.563} C_VEL
LIN {X 0,Y 368.912,Z 489.655,A -85,B 0,C 180,E1 -12640.37,E2 -12640.37} C_VEL
LIN {X 0,Y 368.884,Z 489.657,A -85,B 0,C 180,E1 -12643.616,E2 -12643.616} C_VEL
LIN {X 0,Y 368.906,Z 489.657,A -85,B 0,C 180,E1 -12646.699,E2 -12646.699} C_VEL
LIN {X 0,Y 368.954,Z 489.651,A -85,B 0,C 180,E1 -12649.635,E2 -12649.635} C_VEL
LIN {X 0,Y 368.904,Z 489.656,A -85,B 0,C 180,E1 -12653.144,E2 -12653.144} C_VEL
LIN {X 0,Y 368.903,Z 489.657,A -85,B 0,C 180,E1 -12656.462,E2 -12656.462} C_VEL
LIN {X 0,Y 368.964,Z 489.684,A -85,B 0,C 180,E1 -12657.837,E2 -12657.837} C_VEL
LIN {X 0,Y 373.216,Z 507.391,A -85,B 0,C 180,E1 -12661.609,E2 -12661.609} C_VEL
LIN {X 0,Y 374.25,Z 511.821,A -85,B 0,C 180,E1 -12662.478,E2 -12662.478} C_VEL
LIN {X 0,Y 376.217,Z 519.208,A -85,B 0,C 180,E1 -12663.509,E2 -12663.509} C_VEL
LIN {X 0,Y 376.647,Z 523.165,A -85,B 0,C 180,E1 -12663.928,E2 -12663.928} C_VEL
LIN {X 0,Y 377.341,Z 534.165,A -85,B 0,C 180,E1 -12664.93,E2 -12664.93} C_VEL
LIN {X 0,Y 377.488,Z 548.171,A -85,B 0,C 180,E1 -12665.99,E2 -12665.99} C_VEL
LIN {X 0,Y 378.206,Z 553.878,A -85,B 0,C 180,E1 -12666.174,E2 -12666.174} C_VEL
LIN {X 0,Y 375.328,Z 662.294,A -85,B 0,C 180,E1 -12668.728,E2 -12668.728} C_VEL
LIN {X 0,Y 374.551,Z 677.052,A -85,B 0,C 180,E1 -12669.294,E2 -12669.294} C_VEL
LIN {X 0,Y 373.843,Z 690.789,A -85,B 0,C 180,E1 -12670.046,E2 -12670.046} C_VEL
LIN {X 0,Y 372.909,Z 704.459,A -85,B 0,C 180,E1 -12671.028,E2 -12671.028} C_VEL
LIN {X 0,Y 371.923,Z 716.434,A -85,B 0,C 180,E1 -12672.117,E2 -12672.117} C_VEL
LIN {X 0,Y 370.849,Z 728.596,A -85,B 0,C 180,E1 -12673.485,E2 -12673.485} C_VEL
LIN {X 0,Y 369.952,Z 738.651,A -85,B 0,C 180,E1 -12674.858,E2 -12674.858} C_VEL
LIN {X 0,Y 369.155,Z 748.791,A -85,B 0,C 180,E1 -12676.533,E2 -12676.533} C_VEL
LIN {X 0,Y 368.575,Z 756.949,A -85,B 0,C 180,E1 -12678.172,E2 -12678.172} C_VEL
LIN {X 0,Y 367.997,Z 764.976,A -85,B 0,C 180,E1 -12680.103,E2 -12680.103} C_VEL
LIN {X 0,Y 367.719,Z 770.519,A -85,B 0,C 180,E1 -12681.759,E2 -12681.759} C_VEL
LIN {X 0,Y 367.552,Z 774.816,A -85,B 0,C 180,E1 -12683.412,E2 -12683.412} C_VEL
LIN {X 0,Y 367.459,Z 777.039,A -85,B 0,C 180,E1 -12684.512,E2 -12684.512} C_VEL
LIN {X 0,Y 367.379,Z 780.28,A -85,B 0,C 180,E1 -12686.71,E2 -12686.71} C_VEL
LIN {X 0,Y 367.413,Z 781.427,A -85,B 0,C 180,E1 -12687.808,E2 -12687.808} C_VEL
LIN {X 0,Y 367.458,Z 782.188,A -85,B 0,C 180,E1 -12688.904,E2 -12688.904} C_VEL
LIN {X 0,Y 367.471,Z 782.576,A -85,B 0,C 180,E1 -12690,E2 -12690} C_VEL
LIN {X 0,Y 367.437,Z 782.593,A -85,B 0,C 180,E1 -12691.096,E2 -12691.096} C_VEL
LIN {X 0,Y 367.373,Z 781.527,A -85,B 0,C 180,E1 -12693.29,E2 -12693.29} C_VEL
LIN {X 0,Y 367.451,Z 778.992,A -85,B 0,C 180,E1 -12695.488,E2 -12695.488} C_VEL
LIN {X 0,Y 367.672,Z 774.942,A -85,B 0,C 180,E1 -12697.69,E2 -12697.69} C_VEL
LIN {X 0,Y 367.953,Z 770.788,A -85,B 0,C 180,E1 -12699.344,E2 -12699.344} C_VEL
LIN {X 0,Y 368.385,Z 765.647,A -85,B 0,C 180,E1 -12700.998,E2 -12700.998} C_VEL
LIN {X 0,Y 369.279,Z 758.259,A -85,B 0,C 180,E1 -12702.922,E2 -12702.922} C_VEL
LIN {X 0,Y 370.073,Z 750.645,A -85,B 0,C 180,E1 -12704.546,E2 -12704.546} C_VEL
LIN {X 0,Y 371.236,Z 741.213,A -85,B 0,C 180,E1 -12706.215,E2 -12706.215} C_VEL
LIN {X 0,Y 372.513,Z 730.955,A -85,B 0,C 180,E1 -12707.712,E2 -12707.712} C_VEL
LIN {X 0,Y 373.874,Z 719.747,A -85,B 0,C 180,E1 -12709.063,E2 -12709.063} C_VEL
LIN {X 0,Y 375.318,Z 707.594,A -85,B 0,C 180,E1 -12710.251,E2 -12710.251} C_VEL
LIN {X 0,Y 376.75,Z 693.785,A -85,B 0,C 180,E1 -12711.331,E2 -12711.331} C_VEL
LIN {X 0,Y 377.994,Z 679.52,A -85,B 0,C 180,E1 -12712.189,E2 -12712.189} C_VEL
LIN {X 0,Y 379.19,Z 664.179,A -85,B 0,C 180,E1 -12712.834,E2 -12712.834} C_VEL
LIN {X 0,Y 380.111,Z 641.701,A -85,B 0,C 180,E1 -12713.46,E2 -12713.46} C_VEL
LIN {X 0,Y 383.383,Z 573.652,A -85,B 0,C 180,E1 -12715.268,E2 -12715.268} C_VEL
LIN {X 0,Y 384.308,Z 554.133,A -85,B 0,C 180,E1 -12715.824,E2 -12715.824} C_VEL
LIN {X 0,Y 382.087,Z 540.019,A -85,B 0,C 180,E1 -12716.569,E2 -12716.569} C_VEL
LIN {X 0,Y 379.744,Z 529.231,A -85,B 0,C 180,E1 -12717.247,E2 -12717.247} C_VEL
LIN {X 0,Y 379.962,Z 527.887,A -85,B 0,C 180,E1 -12717.543,E2 -12717.543} C_VEL
LIN {X 0,Y 378.725,Z 520.841,A -85,B 0,C 180,E1 -12719.53,E2 -12719.53} C_VEL
LIN {X 0,Y 376.917,Z 513.41,A -85,B 0,C 180,E1 -12721.996,E2 -12721.996} C_VEL
LIN {X 0,Y 375.184,Z 507.177,A -85,B 0,C 180,E1 -12724.491,E2 -12724.491} C_VEL
LIN {X 0,Y 373.58,Z 502.202,A -85,B 0,C 180,E1 -12727.014,E2 -12727.014} C_VEL
LIN {X 0,Y 372.35,Z 498.902,A -85,B 0,C 180,E1 -12729.298,E2 -12729.298} C_VEL
LIN {X 0,Y 371.596,Z 496.665,A -85,B 0,C 180,E1 -12731.45,E2 -12731.45} C_VEL
LIN {X 0,Y 371.155,Z 495.721,A -85,B 0,C 180,E1 -12732.975,E2 -12732.975} C_VEL
LIN {X 0,Y 370.839,Z 495.152,A -85,B 0,C 180,E1 -12735.476,E2 -12735.476} C_VEL
LIN {X 0,Y 371.046,Z 495.562,A -85,B 0,C 180,E1 -12737.621,E2 -12737.621} C_VEL
LIN {X 0,Y 371.522,Z 496.355,A -85,B 0,C 180,E1 -12739.172,E2 -12739.172} C_VEL
LIN {X 0,Y 372.636,Z 499.726,A -85,B 0,C 180,E1 -12742.385,E2 -12742.385} C_VEL
LIN {X 0,Y 374.004,Z 503.985,A -85,B 0,C 180,E1 -12745.032,E2 -12745.032} C_VEL
LIN {X 0,Y 375.432,Z 508.905,A -85,B 0,C 180,E1 -12747.394,E2 -12747.394} C_VEL
LIN {X 0,Y 376.997,Z 514.862,A -85,B 0,C 180,E1 -12749.779,E2 -12749.779} C_VEL
LIN {X 0,Y 378.245,Z 520.709,A -85,B 0,C 180,E1 -12751.784,E2 -12751.784} C_VEL
LIN {X 0,Y 378.856,Z 526.714,A -85,B 0,C 180,E1 -12753.563,E2 -12753.563} C_VEL
LIN {X 0,Y 376.727,Z 538.249,A -85,B 0,C 180,E1 -12756.283,E2 -12756.283} C_VEL
LIN {X 0,Y 380.6,Z 555.121,A -85,B 0,C 180,E1 -12757.454,E2 -12757.454} C_VEL
LIN {X 0,Y 383.012,Z 570.447,A -85,B 0,C 180,E1 -12758.311,E2 -12758.311} C_VEL
LIN {X 0,Y 382.83,Z 576.306,A -85,B 0,C 180,E1 -12758.512,E2 -12758.512} C_VEL
LIN {X 0,Y 378.991,Z 644.254,A -85,B 0,C 180,E1 -12760.571,E2 -12760.571} C_VEL
LIN {X 0,Y 378.079,Z 659.637,A -85,B 0,C 180,E1 -12761.086,E2 -12761.086} C_VEL
LIN {X 0,Y 376.981,Z 673.953,A -85,B 0,C 180,E1 -12761.804,E2 -12761.804} C_VEL
LIN {X 0,Y 375.894,Z 687.04,A -85,B 0,C 180,E1 -12762.689,E2 -12762.689} C_VEL
LIN {X 0,Y 374.532,Z 699.755,A -85,B 0,C 180,E1 -12763.792,E2 -12763.792} C_VEL
LIN {X 0,Y 373.282,Z 710.828,A -85,B 0,C 180,E1 -12764.996,E2 -12764.996} C_VEL
LIN {X 0,Y 372.234,Z 718.997,A -85,B 0,C 180,E1 -12766.07,E2 -12766.07} C_VEL
LIN {X 0,Y 371.156,Z 727.613,A -85,B 0,C 180,E1 -12767.423,E2 -12767.423} C_VEL
LIN {X 0,Y 370.203,Z 736.095,A -85,B 0,C 180,E1 -12769.056,E2 -12769.056} C_VEL
LIN {X 0,Y 369.33,Z 742.974,A -85,B 0,C 180,E1 -12770.692,E2 -12770.692} C_VEL
LIN {X 0,Y 368.645,Z 748.862,A -85,B 0,C 180,E1 -12772.461,E2 -12772.461} C_VEL
LIN {X 0,Y 368.151,Z 752.761,A -85,B 0,C 180,E1 -12773.973,E2 -12773.973} C_VEL
LIN {X 0,Y 367.903,Z 755.957,A -85,B 0,C 180,E1 -12775.618,E2 -12775.618} C_VEL
LIN {X 0,Y 367.812,Z 757.538,A -85,B 0,C 180,E1 -12776.714,E2 -12776.714} C_VEL
LIN {X 0,Y 367.657,Z 758.65,A -85,B 0,C 180,E1 -12777.809,E2 -12777.809} C_VEL
LIN {X 0,Y 367.537,Z 759.323,A -85,B 0,C 180,E1 -12778.904,E2 -12778.904} C_VEL
LIN {X 0,Y 367.491,Z 759.581,A -85,B 0,C 180,E1 -12780,E2 -12780} C_VEL
LIN {X 0,Y 367.462,Z 759.421,A -85,B 0,C 180,E1 -12781.096,E2 -12781.096} C_VEL
LIN {X 0,Y 367.436,Z 758.792,A -85,B 0,C 180,E1 -12782.192,E2 -12782.192} C_VEL
LIN {X 0,Y 367.44,Z 757.733,A -85,B 0,C 180,E1 -12783.289,E2 -12783.289} C_VEL
LIN {X 0,Y 367.534,Z 756.254,A -85,B 0,C 180,E1 -12784.387,E2 -12784.387} C_VEL
LIN {X 0,Y 367.61,Z 752.797,A -85,B 0,C 180,E1 -12786.202,E2 -12786.202} C_VEL
LIN {X 0,Y 367.793,Z 748.944,A -85,B 0,C 180,E1 -12787.687,E2 -12787.687} C_VEL
LIN {X 0,Y 368.09,Z 743.511,A -85,B 0,C 180,E1 -12789.34,E2 -12789.34} C_VEL
LIN {X 0,Y 368.526,Z 736.664,A -85,B 0,C 180,E1 -12790.994,E2 -12790.994} C_VEL
LIN {X 0,Y 369.261,Z 728.147,A -85,B 0,C 180,E1 -12792.643,E2 -12792.643} C_VEL
LIN {X 0,Y 369.766,Z 719.244,A -85,B 0,C 180,E1 -12794.057,E2 -12794.057} C_VEL
LIN {X 0,Y 370.615,Z 708.907,A -85,B 0,C 180,E1 -12795.396,E2 -12795.396} C_VEL
LIN {X 0,Y 371.498,Z 697.088,A -85,B 0,C 180,E1 -12796.627,E2 -12796.627} C_VEL
LIN {X 0,Y 372.214,Z 685.647,A -85,B 0,C 180,E1 -12797.584,E2 -12797.584} C_VEL
LIN {X 0,Y 372.928,Z 673.036,A -85,B 0,C 180,E1 -12798.401,E2 -12798.401} C_VEL
LIN {X 0,Y 373.551,Z 659.538,A -85,B 0,C 180,E1 -12799.045,E2 -12799.045} C_VEL
LIN {X 0,Y 374.044,Z 645.627,A -85,B 0,C 180,E1 -12799.482,E2 -12799.482} C_VEL
LIN {X 0,Y 376.151,Z 568.426,A -85,B 0,C 180,E1 -12801.431,E2 -12801.431} C_VEL
LIN {X 0,Y 372.057,Z 539.782,A -85,B 0,C 180,E1 -12802.408,E2 -12802.408} C_VEL
LIN {X 0,Y 373.677,Z 522.289,A -85,B 0,C 180,E1 -12805.93,E2 -12805.93} C_VEL
LIN {X 0,Y 374.37,Z 515.158,A -85,B 0,C 180,E1 -12807.383,E2 -12807.383} C_VEL
LIN {X 0,Y 372.992,Z 507.791,A -85,B 0,C 180,E1 -12809.025,E2 -12809.025} C_VEL
LIN {X 0,Y 369.673,Z 493.075,A -85,B 0,C 180,E1 -12812.436,E2 -12812.436} C_VEL
LIN {X 0,Y 368.952,Z 489.654,A -85,B 0,C 180,E1 -12813.278,E2 -12813.278} C_VEL
LIN {X 0,Y 368.905,Z 489.655,A -85,B 0,C 180,E1 -12816.856,E2 -12816.856} C_VEL
LIN {X 0,Y 368.914,Z 489.653,A -85,B 0,C 180,E1 -12820.37,E2 -12820.37} C_VEL
LIN {X 0,Y 368.885,Z 489.663,A -85,B 0,C 180,E1 -12823.616,E2 -12823.616} C_VEL
LIN {X 0,Y 368.887,Z 489.656,A -85,B 0,C 180,E1 -12826.696,E2 -12826.696} C_VEL
LIN {X 0,Y 368.913,Z 489.659,A -85,B 0,C 180,E1 -12829.643,E2 -12829.643} C_VEL
LIN {X 0,Y 368.902,Z 489.656,A -85,B 0,C 180,E1 -12833.144,E2 -12833.144} C_VEL
LIN {X 0,Y 368.9,Z 489.654,A -85,B 0,C 180,E1 -12836.462,E2 -12836.462} C_VEL
LIN {X 0,Y 368.93,Z 489.652,A -85,B 0,C 180,E1 -12839.046,E2 -12839.046} C_VEL
LIN {X 0,Y 368.981,Z 489.651,A -85,B 0,C 180,E1 -12841.564,E2 -12841.564} C_VEL
LIN {X 0,Y 369.001,Z 489.644,A -85,B 0,C 180,E1 -12844.02,E2 -12844.02} C_VEL
LIN {X 0,Y 368.935,Z 489.656,A -85,B 0,C 180,E1 -12847.605,E2 -12847.605} C_VEL
LIN {X 0,Y 368.985,Z 489.646,A -85,B 0,C 180,E1 -12851.107,E2 -12851.107} C_VEL
LIN {X 0,Y 369,Z 489.642,A -85,B 0,C 180,E1 -12854.535,E2 -12854.535} C_VEL
LIN {X 0,Y 369.007,Z 489.643,A -85,B 0,C 180,E1 -12857.907,E2 -12857.907} C_VEL
LIN {X 0,Y 369.231,Z 489.616,A -85,B 0,C 180,E1 -12861.8,E2 -12861.8} C_VEL
LIN {X 0,Y 369.147,Z 489.624,A -85,B 0,C 180,E1 -12864.538,E2 -12864.538} C_VEL
LIN {X 0,Y 369.32,Z 489.605,A -85,B 0,C 180,E1 -12867.819,E2 -12867.819} C_VEL
LIN {X 0,Y 369.46,Z 489.586,A -85,B 0,C 180,E1 -12870,E2 -12870} C_VEL
LIN {X 0,Y 369.321,Z 489.602,A -85,B 0,C 180,E1 -12872.181,E2 -12872.181} C_VEL
LIN {X 0,Y 369.209,Z 489.616,A -85,B 0,C 180,E1 -12876.558,E2 -12876.558} C_VEL
LIN {X 0,Y 369.139,Z 489.625,A -85,B 0,C 180,E1 -12878.761,E2 -12878.761} C_VEL
LIN {X 0,Y 369.007,Z 489.642,A -85,B 0,C 180,E1 -12882.093,E2 -12882.093} C_VEL
LIN {X 0,Y 368.999,Z 489.648,A -85,B 0,C 180,E1 -12885.465,E2 -12885.465} C_VEL
LIN {X 0,Y 368.96,Z 489.649,A -85,B 0,C 180,E1 -12888.894,E2 -12888.894} C_VEL
LIN {X 0,Y 368.937,Z 489.65,A -85,B 0,C 180,E1 -12892.395,E2 -12892.395} C_VEL
LIN {X 0,Y 368.984,Z 489.644,A -85,B 0,C 180,E1 -12895.796,E2 -12895.796} C_VEL
LIN {X 0,Y 368.37,Z 489.723,A -85,B 0,C 180,E1 -12896.707,E2 -12896.707} C_VEL
LIN {X 0,Y 365.508,Z 490.079,A -85,B 0,C 180,E1 -12898.187,E2 -12898.187} C_VEL
LIN {X 0,Y 363.034,Z 490.392,A -85,B 0,C 180,E1 -12899.384,E2 -12899.384} C_VEL
LIN {X 0,Y 361.952,Z 490.521,A -85,B 0,C 180,E1 -12900.311,E2 -12900.311} C_VEL
LIN {X 0,Y 361.855,Z 490.533,A -85,B 0,C 180,E1 -12900.626,E2 -12900.626} C_VEL
LIN {X 0,Y 361.855,Z 490.532,A -85,B 0,C 180,E1 -12904.28,E2 -12904.28} C_VEL
LIN {X 0,Y 361.871,Z 490.535,A -85,B 0,C 180,E1 -12907.224,E2 -12907.224} C_VEL
LIN {X 0,Y 361.838,Z 490.535,A -85,B 0,C 180,E1 -12910.756,E2 -12910.756} C_VEL
LIN {X 0,Y 361.823,Z 490.536,A -85,B 0,C 180,E1 -12914.368,E2 -12914.368} C_VEL
LIN {X 0,Y 361.837,Z 490.538,A -85,B 0,C 180,E1 -12917.568,E2 -12917.568} C_VEL
LIN {X 0,Y 361.871,Z 490.533,A -85,B 0,C 180,E1 -12920.973,E2 -12920.973} C_VEL
LIN {X 0,Y 361.876,Z 490.53,A -85,B 0,C 180,E1 -12924.655,E2 -12924.655} C_VEL
LIN {X 0,Y 361.904,Z 490.554,A -85,B 0,C 180,E1 -12928.621,E2 -12928.621} C_VEL
LIN {X 0,Y 365.561,Z 506.716,A -85,B 0,C 180,E1 -12931.756,E2 -12931.756} C_VEL
LIN {X 0,Y 367.113,Z 514.693,A -85,B 0,C 180,E1 -12933.264,E2 -12933.264} C_VEL
LIN {X 0,Y 366.332,Z 528.358,A -85,B 0,C 180,E1 -12935.64,E2 -12935.64} C_VEL
LIN {X 0,Y 365.262,Z 547.093,A -85,B 0,C 180,E1 -12938.882,E2 -12938.882} C_VEL
LIN {X 0,Y 365.2,Z 548.282,A -85,B 0,C 180,E1 -12939.061,E2 -12939.061} C_VEL
LIN {X 0,Y 368.409,Z 572.972,A -85,B 0,C 180,E1 -12939.852,E2 -12939.852} C_VEL
LIN {X 0,Y 366.255,Z 659.383,A -85,B 0,C 180,E1 -12942.048,E2 -12942.048} C_VEL
LIN {X 0,Y 365.669,Z 672.663,A -85,B 0,C 180,E1 -12942.596,E2 -12942.596} C_VEL
LIN {X 0,Y 365.035,Z 685.531,A -85,B 0,C 180,E1 -12943.358,E2 -12943.358} C_VEL
LIN {X 0,Y 364.297,Z 697.952,A -85,B 0,C 180,E1 -12944.331,E2 -12944.331} C_VEL
LIN {X 0,Y 363.642,Z 709.122,A -85,B 0,C 180,E1 -12945.449,E2 -12945.449} C_VEL
LIN {X 0,Y 362.92,Z 719.33,A -85,B 0,C 180,E1 -12946.705,E2 -12946.705} C_VEL
LIN {X 0,Y 362.117,Z 729.373,A -85,B 0,C 180,E1 -12948.242,E2 -12948.242} C_VEL
LIN {X 0,Y 361.451,Z 738.234,A -85,B 0,C 180,E1 -12949.922,E2 -12949.922} C_VEL
LIN {X 0,Y 360.976,Z 745.274,A -85,B 0,C 180,E1 -12951.604,E2 -12951.604} C_VEL
LIN {X 0,Y 360.719,Z 750.895,A -85,B 0,C 180,E1 -12953.287,E2 -12953.287} C_VEL
LIN {X 0,Y 360.548,Z 755.257,A -85,B 0,C 180,E1 -12954.968,E2 -12954.968} C_VEL
LIN {X 0,Y 360.367,Z 758.477,A -85,B 0,C 180,E1 -12956.646,E2 -12956.646} C_VEL
LIN {X 0,Y 360.322,Z 760.034,A -85,B 0,C 180,E1 -12957.764,E2 -12957.764} C_VEL
LIN {X 0,Y 360.313,Z 761.127,A -85,B 0,C 180,E1 -12958.882,E2 -12958.882} C_VEL
LIN {X 0,Y 360.358,Z 761.806,A -85,B 0,C 180,E1 -12960,E2 -12960} C_VEL
LIN {X 0,Y 360.371,Z 762.035,A -85,B 0,C 180,E1 -12961.117,E2 -12961.117} C_VEL
LIN {X 0,Y 360.416,Z 761.804,A -85,B 0,C 180,E1 -12962.235,E2 -12962.235} C_VEL
LIN {X 0,Y 360.443,Z 761.163,A -85,B 0,C 180,E1 -12963.353,E2 -12963.353} C_VEL
LIN {X 0,Y 360.554,Z 760.091,A -85,B 0,C 180,E1 -12964.472,E2 -12964.472} C_VEL
LIN {X 0,Y 360.843,Z 758.534,A -85,B 0,C 180,E1 -12965.589,E2 -12965.589} C_VEL
LIN {X 0,Y 361.117,Z 755.975,A -85,B 0,C 180,E1 -12966.995,E2 -12966.995} C_VEL
LIN {X 0,Y 361.57,Z 751.101,A -85,B 0,C 180,E1 -12968.946,E2 -12968.946} C_VEL
LIN {X 0,Y 362.326,Z 745.57,A -85,B 0,C 180,E1 -12970.619,E2 -12970.619} C_VEL
LIN {X 0,Y 363.119,Z 738.655,A -85,B 0,C 180,E1 -12972.292,E2 -12972.292} C_VEL
LIN {X 0,Y 364.284,Z 730.022,A -85,B 0,C 180,E1 -12973.955,E2 -12973.955} C_VEL
LIN {X 0,Y 365.532,Z 720.233,A -85,B 0,C 180,E1 -12975.472,E2 -12975.472} C_VEL
LIN {X 0,Y 366.815,Z 709.112,A -85,B 0,C 180,E1 -12976.845,E2 -12976.845} C_VEL
LIN {X 0,Y 367.929,Z 698.094,A -85,B 0,C 180,E1 -12977.94,E2 -12977.94} C_VEL
LIN {X 0,Y 369.11,Z 685.964,A -85,B 0,C 180,E1 -12978.886,E2 -12978.886} C_VEL
LIN {X 0,Y 370.12,Z 673.63,A -85,B 0,C 180,E1 -12979.625,E2 -12979.625} C_VEL
LIN {X 0,Y 370.973,Z 659.259,A -85,B 0,C 180,E1 -12980.227,E2 -12980.227} C_VEL
LIN {X 0,Y 374.842,Z 581.956,A -85,B 0,C 180,E1 -12982.482,E2 -12982.482} C_VEL
LIN {X 0,Y 375.113,Z 573.646,A -85,B 0,C 180,E1 -12982.75,E2 -12982.75} C_VEL
LIN {X 0,Y 373.162,Z 562.156,A -85,B 0,C 180,E1 -12983.387,E2 -12983.387} C_VEL
LIN {X 0,Y 370.642,Z 550.474,A -85,B 0,C 180,E1 -12984.151,E2 -12984.151} C_VEL
LIN {X 0,Y 372.966,Z 528.538,A -85,B 0,C 180,E1 -12988.105,E2 -12988.105} C_VEL
LIN {X 0,Y 373.055,Z 525.622,A -85,B 0,C 180,E1 -12988.685,E2 -12988.685} C_VEL
LIN {X 0,Y 371.778,Z 518.334,A -85,B 0,C 180,E1 -12990.376,E2 -12990.376} C_VEL
LIN {X 0,Y 369.611,Z 510.126,A -85,B 0,C 180,E1 -12992.545,E2 -12992.545} C_VEL
LIN {X 0,Y 366.647,Z 501.589,A -85,B 0,C 180,E1 -12995.103,E2 -12995.103} C_VEL
LIN {X 0,Y 363.754,Z 494.71,A -85,B 0,C 180,E1 -12997.613,E2 -12997.613} C_VEL
LIN {X 0,Y 362.076,Z 491.544,A -85,B 0,C 180,E1 -12999.067,E2 -12999.067} C_VEL
LIN {X 0,Y 361.838,Z 490.54,A -85,B 0,C 180,E1 -12999.514,E2 -12999.514} C_VEL
LIN {X 0,Y 361.837,Z 490.539,A -85,B 0,C 180,E1 -13002.829,E2 -13002.829} C_VEL
LIN {X 0,Y 361.83,Z 490.537,A -85,B 0,C 180,E1 -13005.945,E2 -13005.945} C_VEL
LIN {X 0,Y 361.874,Z 490.531,A -85,B 0,C 180,E1 -13009.238,E2 -13009.238} C_VEL
LIN {X 0,Y 361.87,Z 490.532,A -85,B 0,C 180,E1 -13012.982,E2 -13012.982} C_VEL
LIN {X 0,Y 361.894,Z 490.614,A -85,B 0,C 180,E1 -13016.482,E2 -13016.482} C_VEL
LIN {X 0,Y 362.515,Z 492.736,A -85,B 0,C 180,E1 -13017.123,E2 -13017.123} C_VEL
LIN {X 0,Y 363.61,Z 495.041,A -85,B 0,C 180,E1 -13017.892,E2 -13017.892} C_VEL
LIN {X 0,Y 365.768,Z 504.063,A -85,B 0,C 180,E1 -13019.842,E2 -13019.842} C_VEL
LIN {X 0,Y 369.071,Z 515.121,A -85,B 0,C 180,E1 -13021.897,E2 -13021.897} C_VEL
LIN {X 0,Y 370.878,Z 522.285,A -85,B 0,C 180,E1 -13022.953,E2 -13022.953} C_VEL
LIN {X 0,Y 371.281,Z 526.257,A -85,B 0,C 180,E1 -13023.389,E2 -13023.389} C_VEL
LIN {X 0,Y 371.761,Z 536.722,A -85,B 0,C 180,E1 -13024.377,E2 -13024.377} C_VEL
LIN {X 0,Y 371.713,Z 554.236,A -85,B 0,C 180,E1 -13025.731,E2 -13025.731} C_VEL
LIN {X 0,Y 371.25,Z 558.761,A -85,B 0,C 180,E1 -13025.971,E2 -13025.971} C_VEL
LIN {X 0,Y 368.419,Z 662.661,A -85,B 0,C 180,E1 -13028.493,E2 -13028.493} C_VEL
LIN {X 0,Y 367.611,Z 677.229,A -85,B 0,C 180,E1 -13029.068,E2 -13029.068} C_VEL
LIN {X 0,Y 366.892,Z 690.816,A -85,B 0,C 180,E1 -13029.83,E2 -13029.83} C_VEL
LIN {X 0,Y 365.941,Z 704.193,A -85,B 0,C 180,E1 -13030.81,E2 -13030.81} C_VEL
LIN {X 0,Y 364.958,Z 716.093,A -85,B 0,C 180,E1 -13031.909,E2 -13031.909} C_VEL
LIN {X 0,Y 363.844,Z 728.285,A -85,B 0,C 180,E1 -13033.302,E2 -13033.302} C_VEL
LIN {X 0,Y 362.675,Z 741.375,A -85,B 0,C 180,E1 -13035.122,E2 -13035.122} C_VEL
LIN {X 0,Y 362.098,Z 749.928,A -85,B 0,C 180,E1 -13036.532,E2 -13036.532} C_VEL
LIN {X 0,Y 361.521,Z 758.393,A -85,B 0,C 180,E1 -13038.222,E2 -13038.222} C_VEL
LIN {X 0,Y 360.969,Z 765.232,A -85,B 0,C 180,E1 -13039.908,E2 -13039.908} C_VEL
LIN {X 0,Y 360.668,Z 770.649,A -85,B 0,C 180,E1 -13041.596,E2 -13041.596} C_VEL
LIN {X 0,Y 360.481,Z 774.843,A -85,B 0,C 180,E1 -13043.282,E2 -13043.282} C_VEL
LIN {X 0,Y 360.382,Z 777.016,A -85,B 0,C 180,E1 -13044.404,E2 -13044.404} C_VEL
LIN {X 0,Y 360.355,Z 778.742,A -85,B 0,C 180,E1 -13045.526,E2 -13045.526} C_VEL
LIN {X 0,Y 360.315,Z 781.074,A -85,B 0,C 180,E1 -13047.764,E2 -13047.764} C_VEL
LIN {X 0,Y 360.361,Z 781.888,A -85,B 0,C 180,E1 -13048.883,E2 -13048.883} C_VEL
LIN {X 0,Y 360.376,Z 782.315,A -85,B 0,C 180,E1 -13050,E2 -13050} C_VEL
LIN {X 0,Y 360.338,Z 782.367,A -85,B 0,C 180,E1 -13051.118,E2 -13051.118} C_VEL
LIN {X 0,Y 360.292,Z 781.366,A -85,B 0,C 180,E1 -13053.355,E2 -13053.355} C_VEL
LIN {X 0,Y 360.359,Z 778.897,A -85,B 0,C 180,E1 -13055.596,E2 -13055.596} C_VEL
LIN {X 0,Y 360.621,Z 774.912,A -85,B 0,C 180,E1 -13057.841,E2 -13057.841} C_VEL
LIN {X 0,Y 360.913,Z 770.83,A -85,B 0,C 180,E1 -13059.528,E2 -13059.528} C_VEL
LIN {X 0,Y 361.387,Z 765.768,A -85,B 0,C 180,E1 -13061.214,E2 -13061.214} C_VEL
LIN {X 0,Y 362.339,Z 758.463,A -85,B 0,C 180,E1 -13063.174,E2 -13063.174} C_VEL
LIN {X 0,Y 363.231,Z 750.811,A -85,B 0,C 180,E1 -13064.855,E2 -13064.855} C_VEL
LIN {X 0,Y 364.418,Z 741.638,A -85,B 0,C 180,E1 -13066.527,E2 -13066.527} C_VEL
LIN {X 0,Y 365.898,Z 730.538,A -85,B 0,C 180,E1 -13068.187,E2 -13068.187} C_VEL
LIN {X 0,Y 367.383,Z 719.307,A -85,B 0,C 180,E1 -13069.559,E2 -13069.559} C_VEL
LIN {X 0,Y 368.879,Z 707.482,A -85,B 0,C 180,E1 -13070.735,E2 -13070.735} C_VEL
LIN {X 0,Y 370.388,Z 693.931,A -85,B 0,C 180,E1 -13071.819,E2 -13071.819} C_VEL
LIN {X 0,Y 371.671,Z 680.351,A -85,B 0,C 180,E1 -13072.661,E2 -13072.661} C_VEL
LIN {X 0,Y 372.933,Z 665.772,A -85,B 0,C 180,E1 -13073.313,E2 -13073.313} C_VEL
LIN {X 0,Y 373.731,Z 648.188,A -85,B 0,C 180,E1 -13073.848,E2 -13073.848} C_VEL
LIN {X 0,Y 377.203,Z 580.975,A -85,B 0,C 180,E1 -13075.682,E2 -13075.682} C_VEL
LIN {X 0,Y 378.544,Z 555.294,A -85,B 0,C 180,E1 -13076.437,E2 -13076.437} C_VEL
LIN {X 0,Y 376.732,Z 543.042,A -85,B 0,C 180,E1 -13077.108,E2 -13077.108} C_VEL
LIN {X 0,Y 374.262,Z 531.53,A -85,B 0,C 180,E1 -13077.872,E2 -13077.872} C_VEL
LIN {X 0,Y 373.466,Z 529.546,A -85,B 0,C 180,E1 -13078.064,E2 -13078.064} C_VEL
LIN {X 0,Y 372.26,Z 522.971,A -85,B 0,C 180,E1 -13080.025,E2 -13080.025} C_VEL
LIN {X 0,Y 370.56,Z 516.007,A -85,B 0,C 180,E1 -13082.461,E2 -13082.461} C_VEL
LIN {X 0,Y 368.926,Z 510.063,A -85,B 0,C 180,E1 -13085.001,E2 -13085.001} C_VEL
LIN {X 0,Y 367.35,Z 505.142,A -85,B 0,C 180,E1 -13087.75,E2 -13087.75} C_VEL
LIN {X 0,Y 366.33,Z 502.402,A -85,B 0,C 180,E1 -13089.879,E2 -13089.879} C_VEL
LIN {X 0,Y 365.641,Z 500.279,A -85,B 0,C 180,E1 -13092.279,E2 -13092.279} C_VEL
LIN {X 0,Y 365.189,Z 499.438,A -85,B 0,C 180,E1 -13094.597,E2 -13094.597} C_VEL
LIN {X 0,Y 365.261,Z 499.554,A -85,B 0,C 180,E1 -13096.984,E2 -13096.984} C_VEL
LIN {X 0,Y 365.783,Z 500.563,A -85,B 0,C 180,E1 -13099.212,E2 -13099.212} C_VEL
LIN {X 0,Y 366.722,Z 503.541,A -85,B 0,C 180,E1 -13102.174,E2 -13102.174} C_VEL
LIN {X 0,Y 368.179,Z 508.165,A -85,B 0,C 180,E1 -13105.166,E2 -13105.166} C_VEL
LIN {X 0,Y 369.664,Z 513.727,A -85,B 0,C 180,E1 -13107.837,E2 -13107.837} C_VEL
LIN {X 0,Y 371.282,Z 520.627,A -85,B 0,C 180,E1 -13110.545,E2 -13110.545} C_VEL
LIN {X 0,Y 372.295,Z 526.614,A -85,B 0,C 180,E1 -13112.53,E2 -13112.53} C_VEL
LIN {X 0,Y 372.375,Z 529.521,A -85,B 0,C 180,E1 -13113.369,E2 -13113.369} C_VEL
LIN {X 0,Y 370.649,Z 538.298,A -85,B 0,C 180,E1 -13115.461,E2 -13115.461} C_VEL
LIN {X 0,Y 374.636,Z 555.075,A -85,B 0,C 180,E1 -13116.721,E2 -13116.721} C_VEL
LIN {X 0,Y 376.829,Z 568.75,A -85,B 0,C 180,E1 -13117.558,E2 -13117.558} C_VEL
LIN {X 0,Y 377.265,Z 573.21,A -85,B 0,C 180,E1 -13117.789,E2 -13117.789} C_VEL
LIN {X 0,Y 372.042,Z 657.931,A -85,B 0,C 180,E1 -13120.481,E2 -13120.481} C_VEL
LIN {X 0,Y 371.086,Z 670.507,A -85,B 0,C 180,E1 -13121.075,E2 -13121.075} C_VEL
LIN {X 0,Y 369.929,Z 682.9,A -85,B 0,C 180,E1 -13121.861,E2 -13121.861} C_VEL
LIN {X 0,Y 368.587,Z 695.667,A -85,B 0,C 180,E1 -13122.907,E2 -13122.907} C_VEL
LIN {X 0,Y 367.101,Z 707.818,A -85,B 0,C 180,E1 -13124.168,E2 -13124.168} C_VEL
LIN {X 0,Y 365.7,Z 718.461,A -85,B 0,C 180,E1 -13125.532,E2 -13125.532} C_VEL
LIN {X 0,Y 364.53,Z 727.221,A -85,B 0,C 180,E1 -13126.907,E2 -13126.907} C_VEL
LIN {X 0,Y 363.512,Z 735.792,A -85,B 0,C 180,E1 -13128.57,E2 -13128.57} C_VEL
LIN {X 0,Y 362.493,Z 742.751,A -85,B 0,C 180,E1 -13130.233,E2 -13130.233} C_VEL
LIN {X 0,Y 361.693,Z 749.187,A -85,B 0,C 180,E1 -13132.183,E2 -13132.183} C_VEL
LIN {X 0,Y 361.129,Z 753.382,A -85,B 0,C 180,E1 -13133.855,E2 -13133.855} C_VEL
LIN {X 0,Y 360.837,Z 756.466,A -85,B 0,C 180,E1 -13135.532,E2 -13135.532} C_VEL
LIN {X 0,Y 360.747,Z 757.967,A -85,B 0,C 180,E1 -13136.649,E2 -13136.649} C_VEL
LIN {X 0,Y 360.585,Z 759.005,A -85,B 0,C 180,E1 -13137.766,E2 -13137.766} C_VEL
LIN {X 0,Y 360.459,Z 759.633,A -85,B 0,C 180,E1 -13138.883,E2 -13138.883} C_VEL
LIN {X 0,Y 360.395,Z 759.846,A -85,B 0,C 180,E1 -13140,E2 -13140} C_VEL
LIN {X 0,Y 360.363,Z 759.607,A -85,B 0,C 180,E1 -13141.117,E2 -13141.117} C_VEL
LIN {X 0,Y 360.337,Z 758.915,A -85,B 0,C 180,E1 -13142.236,E2 -13142.236} C_VEL
LIN {X 0,Y 360.358,Z 757.803,A -85,B 0,C 180,E1 -13143.354,E2 -13143.354} C_VEL
LIN {X 0,Y 360.464,Z 755.291,A -85,B 0,C 180,E1 -13145.033,E2 -13145.033} C_VEL
LIN {X 0,Y 360.584,Z 751.718,A -85,B 0,C 180,E1 -13146.716,E2 -13146.716} C_VEL
LIN {X 0,Y 360.827,Z 746.991,A -85,B 0,C 180,E1 -13148.4,E2 -13148.4} C_VEL
LIN {X 0,Y 361.208,Z 740.981,A -85,B 0,C 180,E1 -13150.085,E2 -13150.085} C_VEL
LIN {X 0,Y 361.739,Z 733.468,A -85,B 0,C 180,E1 -13151.771,E2 -13151.771} C_VEL
LIN {X 0,Y 362.326,Z 725.827,A -85,B 0,C 180,E1 -13153.174,E2 -13153.174} C_VEL
LIN {X 0,Y 363.062,Z 715.587,A -85,B 0,C 180,E1 -13154.718,E2 -13154.718} C_VEL
LIN {X 0,Y 363.854,Z 705.354,A -85,B 0,C 180,E1 -13155.977,E2 -13155.977} C_VEL
LIN {X 0,Y 364.771,Z 694.171,A -85,B 0,C 180,E1 -13157.087,E2 -13157.087} C_VEL
LIN {X 0,Y 365.51,Z 681.904,A -85,B 0,C 180,E1 -13158.062,E2 -13158.062} C_VEL
LIN {X 0,Y 366.171,Z 669.469,A -85,B 0,C 180,E1 -13158.825,E2 -13158.825} C_VEL
LIN {X 0,Y 366.801,Z 655.149,A -85,B 0,C 180,E1 -13159.445,E2 -13159.445} C_VEL
LIN {X 0,Y 367.959,Z 618.196,A -85,B 0,C 180,E1 -13160.433,E2 -13160.433} C_VEL
LIN {X 0,Y 369.339,Z 569.353,A -85,B 0,C 180,E1 -13161.71,E2 -13161.71} C_VEL
LIN {X 0,Y 365.176,Z 539.607,A -85,B 0,C 180,E1 -13162.759,E2 -13162.759} C_VEL
LIN {X 0,Y 366.77,Z 523.062,A -85,B 0,C 180,E1 -13166.15,E2 -13166.15} C_VEL
LIN {X 0,Y 367.403,Z 516.172,A -85,B 0,C 180,E1 -13167.582,E2 -13167.582} C_VEL
LIN {X 0,Y 365.668,Z 507.438,A -85,B 0,C 180,E1 -13169.572,E2 -13169.572} C_VEL
LIN {X 0,Y 361.965,Z 490.786,A -85,B 0,C 180,E1 -13173.523,E2 -13173.523} C_VEL
LIN {X 0,Y 361.929,Z 490.529,A -85,B 0,C 180,E1 -13173.775,E2 -13173.775} C_VEL
LIN {X 0,Y 361.874,Z 490.533,A -85,B 0,C 180,E1 -13177.224,E2 -13177.224} C_VEL
LIN {X 0,Y 361.838,Z 490.534,A -85,B 0,C 180,E1 -13180.755,E2 -13180.755} C_VEL
LIN {X 0,Y 361.819,Z 490.537,A -85,B 0,C 180,E1 -13184.368,E2 -13184.368} C_VEL
LIN {X 0,Y 361.838,Z 490.541,A -85,B 0,C 180,E1 -13187.568,E2 -13187.568} C_VEL
LIN {X 0,Y 361.87,Z 490.531,A -85,B 0,C 180,E1 -13190.973,E2 -13190.973} C_VEL
LIN {X 0,Y 361.876,Z 490.53,A -85,B 0,C 180,E1 -13194.655,E2 -13194.655} C_VEL
LIN {X 0,Y 361.841,Z 490.534,A -85,B 0,C 180,E1 -13198.371,E2 -13198.371} C_VEL
LIN {X 0,Y 361.902,Z 490.527,A -85,B 0,C 180,E1 -13200.955,E2 -13200.955} C_VEL
LIN {X 0,Y 361.956,Z 490.526,A -85,B 0,C 180,E1 -13203.475,E2 -13203.475} C_VEL
LIN {X 0,Y 361.892,Z 490.53,A -85,B 0,C 180,E1 -13207.145,E2 -13207.145} C_VEL
LIN {X 0,Y 361.923,Z 490.524,A -85,B 0,C 180,E1 -13210.724,E2 -13210.724} C_VEL
LIN {X 0,Y 361.948,Z 490.521,A -85,B 0,C 180,E1 -13214.226,E2 -13214.226} C_VEL
LIN {X 0,Y 362,Z 490.514,A -85,B 0,C 180,E1 -13216.528,E2 -13216.528} C_VEL
LIN {X 0,Y 362.033,Z 490.512,A -85,B 0,C 180,E1 -13219.938,E2 -13219.938} C_VEL
LIN {X 0,Y 362.153,Z 490.495,A -85,B 0,C 180,E1 -13222.193,E2 -13222.193} C_VEL
LIN {X 0,Y 362.12,Z 490.499,A -85,B 0,C 180,E1 -13224.431,E2 -13224.431} C_VEL
LIN {X 0,Y 362.284,Z 490.482,A -85,B 0,C 180,E1 -13227.776,E2 -13227.776} C_VEL
LIN {X 0,Y 362.43,Z 490.462,A -85,B 0,C 180,E1 -13230,E2 -13230} C_VEL
LIN {X 0,Y 362.285,Z 490.479,A -85,B 0,C 180,E1 -13232.223,E2 -13232.223} C_VEL
LIN {X 0,Y 362.172,Z 490.493,A -85,B 0,C 180,E1 -13236.686,E2 -13236.686} C_VEL
LIN {X 0,Y 362.075,Z 490.506,A -85,B 0,C 180,E1 -13238.933,E2 -13238.933} C_VEL
LIN {X 0,Y 361.962,Z 490.519,A -85,B 0,C 180,E1 -13242.332,E2 -13242.332} C_VEL
LIN {X 0,Y 361.963,Z 490.519,A -85,B 0,C 180,E1 -13244.62,E2 -13244.62} C_VEL
LIN {X 0,Y 361.957,Z 490.52,A -85,B 0,C 180,E1 -13248.099,E2 -13248.099} C_VEL
LIN {X 0,Y 361.894,Z 490.531,A -85,B 0,C 180,E1 -13251.653,E2 -13251.653} C_VEL
LIN {X 0,Y 361.93,Z 490.529,A -85,B 0,C 180,E1 -13255.29,E2 -13255.29} C_VEL
LIN {X 0,Y 361.909,Z 490.528,A -85,B 0,C 180,E1 -13257.779,E2 -13257.779} C_VEL
LIN {X 0,Y 361.855,Z 490.533,A -85,B 0,C 180,E1 -13260.626,E2 -13260.626} C_VEL
LIN {X 0,Y 361.161,Z 490.623,A -85,B 0,C 180,E1 -13261.555,E2 -13261.555} C_VEL
LIN {X 0,Y 358.293,Z 490.98,A -85,B 0,C 180,E1 -13263.066,E2 -13263.066} C_VEL
LIN {X 0,Y 355.894,Z 491.277,A -85,B 0,C 180,E1 -13264.289,E2 -13264.289} C_VEL
LIN {X 0,Y 354.887,Z 491.405,A -85,B 0,C 180,E1 -13265.235,E2 -13265.235} C_VEL
LIN {X 0,Y 354.817,Z 491.411,A -85,B 0,C 180,E1 -13265.555,E2 -13265.555} C_VEL
LIN {X 0,Y 354.825,Z 491.413,A -85,B 0,C 180,E1 -13269.424,E2 -13269.424} C_VEL
LIN {X 0,Y 354.79,Z 491.414,A -85,B 0,C 180,E1 -13272.867,E2 -13272.867} C_VEL
LIN {X 0,Y 354.782,Z 491.413,A -85,B 0,C 180,E1 -13276.106,E2 -13276.106} C_VEL
LIN {X 0,Y 354.789,Z 491.417,A -85,B 0,C 180,E1 -13279.179,E2 -13279.179} C_VEL
LIN {X 0,Y 354.809,Z 491.41,A -85,B 0,C 180,E1 -13282.403,E2 -13282.403} C_VEL
LIN {X 0,Y 354.814,Z 491.412,A -85,B 0,C 180,E1 -13284.941,E2 -13284.941} C_VEL
LIN {X 0,Y 354.879,Z 491.48,A -85,B 0,C 180,E1 -13288.333,E2 -13288.333} C_VEL
LIN {X 0,Y 358.665,Z 508.251,A -85,B 0,C 180,E1 -13291.63,E2 -13291.63} C_VEL
LIN {X 0,Y 360.132,Z 515.518,A -85,B 0,C 180,E1 -13293.017,E2 -13293.017} C_VEL
LIN {X 0,Y 359.803,Z 524.17,A -85,B 0,C 180,E1 -13294.55,E2 -13294.55} C_VEL
LIN {X 0,Y 358.499,Z 544.61,A -85,B 0,C 180,E1 -13298.132,E2 -13298.132} C_VEL
LIN {X 0,Y 358.283,Z 548.174,A -85,B 0,C 180,E1 -13298.751,E2 -13298.751} C_VEL
LIN {X 0,Y 361.514,Z 573.502,A -85,B 0,C 180,E1 -13299.591,E2 -13299.591} C_VEL
LIN {X 0,Y 359.279,Z 660.108,A -85,B 0,C 180,E1 -13301.872,E2 -13301.872} C_VEL
LIN {X 0,Y 358.66,Z 673.805,A -85,B 0,C 180,E1 -13302.466,E2 -13302.466} C_VEL
LIN {X 0,Y 357.954,Z 687.458,A -85,B 0,C 180,E1 -13303.313,E2 -13303.313} C_VEL
LIN {X 0,Y 357.169,Z 699.43,A -85,B 0,C 180,E1 -13304.303,E2 -13304.303} C_VEL
LIN {X 0,Y 356.518,Z 710.388,A -85,B 0,C 180,E1 -13305.443,E2 -13305.443} C_VEL
LIN {X 0,Y 355.877,Z 719.375,A -85,B 0,C 180,E1 -13306.583,E2 -13306.583} C_VEL
LIN {X 0,Y 355.103,Z 728.634,A -85,B 0,C 180,E1 -13308.006,E2 -13308.006} C_VEL
LIN {X 0,Y 354.419,Z 737.688,A -85,B 0,C 180,E1 -13309.72,E2 -13309.72} C_VEL
LIN {X 0,Y 353.941,Z 744.91,A -85,B 0,C 180,E1 -13311.436,E2 -13311.436} C_VEL
LIN {X 0,Y 353.637,Z 750.653,A -85,B 0,C 180,E1 -13313.152,E2 -13313.152} C_VEL
LIN {X 0,Y 353.449,Z 755.126,A -85,B 0,C 180,E1 -13314.866,E2 -13314.866} C_VEL
LIN {X 0,Y 353.292,Z 758.448,A -85,B 0,C 180,E1 -13316.579,E2 -13316.579} C_VEL
LIN {X 0,Y 353.228,Z 760.089,A -85,B 0,C 180,E1 -13317.719,E2 -13317.719} C_VEL
LIN {X 0,Y 353.214,Z 761.23,A -85,B 0,C 180,E1 -13318.86,E2 -13318.86} C_VEL
LIN {X 0,Y 353.26,Z 761.95,A -85,B 0,C 180,E1 -13320,E2 -13320} C_VEL
LIN {X 0,Y 353.275,Z 762.255,A -85,B 0,C 180,E1 -13321.14,E2 -13321.14} C_VEL
LIN {X 0,Y 353.322,Z 762.082,A -85,B 0,C 180,E1 -13322.28,E2 -13322.28} C_VEL
LIN {X 0,Y 353.362,Z 761.488,A -85,B 0,C 180,E1 -13323.421,E2 -13323.421} C_VEL
LIN {X 0,Y 353.5,Z 760.477,A -85,B 0,C 180,E1 -13324.561,E2 -13324.561} C_VEL
LIN {X 0,Y 353.803,Z 758.982,A -85,B 0,C 180,E1 -13325.7,E2 -13325.7} C_VEL
LIN {X 0,Y 354.139,Z 755.902,A -85,B 0,C 180,E1 -13327.411,E2 -13327.411} C_VEL
LIN {X 0,Y 354.587,Z 751.714,A -85,B 0,C 180,E1 -13329.123,E2 -13329.123} C_VEL
LIN {X 0,Y 355.39,Z 746.317,A -85,B 0,C 180,E1 -13330.828,E2 -13330.828} C_VEL
LIN {X 0,Y 356.241,Z 739.556,A -85,B 0,C 180,E1 -13332.534,E2 -13332.534} C_VEL
LIN {X 0,Y 357.477,Z 731.069,A -85,B 0,C 180,E1 -13334.226,E2 -13334.226} C_VEL
LIN {X 0,Y 358.67,Z 722.379,A -85,B 0,C 180,E1 -13335.63,E2 -13335.63} C_VEL
LIN {X 0,Y 360.042,Z 711.87,A -85,B 0,C 180,E1 -13337.026,E2 -13337.026} C_VEL
LIN {X 0,Y 361.36,Z 700.049,A -85,B 0,C 180,E1 -13338.277,E2 -13338.277} C_VEL
LIN {X 0,Y 362.575,Z 688.449,A -85,B 0,C 180,E1 -13339.24,E2 -13339.24} C_VEL
LIN {X 0,Y 363.712,Z 675.497,A -85,B 0,C 180,E1 -13340.059,E2 -13340.059} C_VEL
LIN {X 0,Y 364.655,Z 662.126,A -85,B 0,C 180,E1 -13340.667,E2 -13340.667} C_VEL
LIN {X 0,Y 369.361,Z 576.012,A -85,B 0,C 180,E1 -13343.297,E2 -13343.297} C_VEL
LIN {X 0,Y 367.747,Z 565.274,A -85,B 0,C 180,E1 -13343.908,E2 -13343.908} C_VEL
LIN {X 0,Y 364.624,Z 550.831,A -85,B 0,C 180,E1 -13344.899,E2 -13344.899} C_VEL
LIN {X 0,Y 367.002,Z 530.718,A -85,B 0,C 180,E1 -13348.603,E2 -13348.603} C_VEL
LIN {X 0,Y 366.707,Z 526.397,A -85,B 0,C 180,E1 -13349.543,E2 -13349.543} C_VEL
LIN {X 0,Y 365.296,Z 519.457,A -85,B 0,C 180,E1 -13351.296,E2 -13351.296} C_VEL
LIN {X 0,Y 363.019,Z 511.228,A -85,B 0,C 180,E1 -13353.646,E2 -13353.646} C_VEL
LIN {X 0,Y 360.728,Z 504.77,A -85,B 0,C 180,E1 -13355.767,E2 -13355.767} C_VEL
LIN {X 0,Y 358.595,Z 499.439,A -85,B 0,C 180,E1 -13357.841,E2 -13357.841} C_VEL
LIN {X 0,Y 356.686,Z 495.389,A -85,B 0,C 180,E1 -13359.786,E2 -13359.786} C_VEL
LIN {X 0,Y 354.907,Z 492.126,A -85,B 0,C 180,E1 -13361.826,E2 -13361.826} C_VEL
LIN {X 0,Y 354.795,Z 491.413,A -85,B 0,C 180,E1 -13362.337,E2 -13362.337} C_VEL
LIN {X 0,Y 354.795,Z 491.412,A -85,B 0,C 180,E1 -13365.489,E2 -13365.489} C_VEL
LIN {X 0,Y 354.825,Z 491.409,A -85,B 0,C 180,E1 -13369.184,E2 -13369.184} C_VEL
LIN {X 0,Y 354.81,Z 491.411,A -85,B 0,C 180,E1 -13372.402,E2 -13372.402} C_VEL
LIN {X 0,Y 354.826,Z 491.529,A -85,B 0,C 180,E1 -13373.651,E2 -13373.651} C_VEL
LIN {X 0,Y 355.951,Z 494.438,A -85,B 0,C 180,E1 -13375.069,E2 -13375.069} C_VEL
LIN {X 0,Y 356.951,Z 495.648,A -85,B 0,C 180,E1 -13375.785,E2 -13375.785} C_VEL
LIN {X 0,Y 359.047,Z 499.469,A -85,B 0,C 180,E1 -13377.318,E2 -13377.318} C_VEL
LIN {X 0,Y 361.076,Z 508.248,A -85,B 0,C 180,E1 -13379.317,E2 -13379.317} C_VEL
